LIN {X 0,Y 513.803,Z 636.667,A -85,B 0,C 180,E1 25249.021,E2 25249.021} C_VEL
LIN {X 0,Y 513.812,Z 636.664,A -85,B 0,C 180,E1 25245.53,E2 25245.53} C_VEL
LIN {X 0,Y 513.773,Z 636.668,A -85,B 0,C 180,E1 25244.581,E2 25244.581} C_VEL
LIN {X 0,Y 521.434,Z 663.371,A -85,B 0,C 180,E1 25241.928,E2 25241.928} C_VEL
LIN {X 0,Y 524.036,Z 673.946,A -85,B 0,C 180,E1 25240.926,E2 25240.926} C_VEL
LIN {X 0,Y 522.658,Z 718.938,A -85,B 0,C 180,E1 25237.269,E2 25237.269} C_VEL
LIN {X 0,Y 521.288,Z 761.013,A -85,B 0,C 180,E1 25233.85,E2 25233.85} C_VEL
LIN {X 0,Y 519.996,Z 802.226,A -85,B 0,C 180,E1 25230.503,E2 25230.503} C_VEL
LIN {X 0,Y 519.096,Z 834.822,A -85,B 0,C 180,E1 25227.908,E2 25227.908} C_VEL
LIN {X 0,Y 519.16,Z 847.578,A -85,B 0,C 180,E1 25227.692,E2 25227.692} C_VEL
LIN {X 0,Y 517.25,Z 978.274,A -85,B 0,C 180,E1 25225.563,E2 25225.563} C_VEL
LIN {X 0,Y 517.072,Z 994.179,A -85,B 0,C 180,E1 25225.113,E2 25225.113} C_VEL
LIN {X 0,Y 516.715,Z 1010.152,A -85,B 0,C 180,E1 25224.46,E2 25224.46} C_VEL
LIN {X 0,Y 516.263,Z 1025.12,A -85,B 0,C 180,E1 25223.632,E2 25223.632} C_VEL
LIN {X 0,Y 515.746,Z 1039.216,A -85,B 0,C 180,E1 25222.636,E2 25222.636} C_VEL
LIN {X 0,Y 515.163,Z 1052.41,A -85,B 0,C 180,E1 25221.458,E2 25221.458} C_VEL
LIN {X 0,Y 514.609,Z 1064.521,A -85,B 0,C 180,E1 25220.112,E2 25220.112} C_VEL
LIN {X 0,Y 514.083,Z 1075.294,A -85,B 0,C 180,E1 25218.598,E2 25218.598} C_VEL
LIN {X 0,Y 513.701,Z 1083.812,A -85,B 0,C 180,E1 25217.089,E2 25217.089} C_VEL
LIN {X 0,Y 513.406,Z 1091.297,A -85,B 0,C 180,E1 25215.356,E2 25215.356} C_VEL
LIN {X 0,Y 513.242,Z 1096.383,A -85,B 0,C 180,E1 25213.747,E2 25213.747} C_VEL
LIN {X 0,Y 513.159,Z 1100.181,A -85,B 0,C 180,E1 25211.917,E2 25211.917} C_VEL
LIN {X 0,Y 513.19,Z 1101.973,A -85,B 0,C 180,E1 25210.21,E2 25210.21} C_VEL
LIN {X 0,Y 513.311,Z 1102.014,A -85,B 0,C 180,E1 25208.398,E2 25208.398} C_VEL
LIN {X 0,Y 513.529,Z 1100.384,A -85,B 0,C 180,E1 25206.706,E2 25206.706} C_VEL
LIN {X 0,Y 513.882,Z 1096.719,A -85,B 0,C 180,E1 25204.909,E2 25204.909} C_VEL
LIN {X 0,Y 514.348,Z 1091.471,A -85,B 0,C 180,E1 25203.229,E2 25203.229} C_VEL
LIN {X 0,Y 514.952,Z 1084.154,A -85,B 0,C 180,E1 25201.555,E2 25201.555} C_VEL
LIN {X 0,Y 515.626,Z 1075.956,A -85,B 0,C 180,E1 25200.109,E2 25200.109} C_VEL
LIN {X 0,Y 516.42,Z 1065.525,A -85,B 0,C 180,E1 25198.666,E2 25198.666} C_VEL
LIN {X 0,Y 517.22,Z 1054.065,A -85,B 0,C 180,E1 25197.394,E2 25197.394} C_VEL
LIN {X 0,Y 518.038,Z 1040.208,A -85,B 0,C 180,E1 25196.18,E2 25196.18} C_VEL
LIN {X 0,Y 518.657,Z 1026.603,A -85,B 0,C 180,E1 25195.243,E2 25195.243} C_VEL
LIN {X 0,Y 519.137,Z 1013.166,A -85,B 0,C 180,E1 25194.527,E2 25194.527} C_VEL
LIN {X 0,Y 519.486,Z 999.878,A -85,B 0,C 180,E1 25193.98,E2 25193.98} C_VEL
LIN {X 0,Y 519.702,Z 985.077,A -85,B 0,C 180,E1 25193.528,E2 25193.528} C_VEL
LIN {X 0,Y 520.188,Z 943.34,A -85,B 0,C 180,E1 25192.784,E2 25192.784} C_VEL
LIN {X 0,Y 522.879,Z 843.141,A -85,B 0,C 180,E1 25191.004,E2 25191.004} C_VEL
LIN {X 0,Y 523.363,Z 837.807,A -85,B 0,C 180,E1 25190.596,E2 25190.596} C_VEL
LIN {X 0,Y 524.872,Z 795.815,A -85,B 0,C 180,E1 25187.231,E2 25187.231} C_VEL
LIN {X 0,Y 526.347,Z 751.412,A -85,B 0,C 180,E1 25183.726,E2 25183.726} C_VEL
LIN {X 0,Y 527.629,Z 711.745,A -85,B 0,C 180,E1 25180.63,E2 25180.63} C_VEL
LIN {X 0,Y 528.648,Z 676.247,A -85,B 0,C 180,E1 25177.888,E2 25177.888} C_VEL
LIN {X 0,Y 524.106,Z 661.406,A -85,B 0,C 180,E1 25176.306,E2 25176.306} C_VEL
LIN {X 0,Y 518.577,Z 647.638,A -85,B 0,C 180,E1 25174.654,E2 25174.654} C_VEL
LIN {X 0,Y 515.244,Z 640.334,A -85,B 0,C 180,E1 25173.705,E2 25173.705} C_VEL
LIN {X 0,Y 513.838,Z 636.878,A -85,B 0,C 180,E1 25173.27,E2 25173.27} C_VEL
LIN {X 0,Y 513.821,Z 636.667,A -85,B 0,C 180,E1 25169.732,E2 25169.732} C_VEL
LIN {X 0,Y 513.795,Z 636.668,A -85,B 0,C 180,E1 25166.178,E2 25166.178} C_VEL
LIN {X 0,Y 513.774,Z 636.672,A -85,B 0,C 180,E1 25162.744,E2 25162.744} C_VEL
LIN {X 0,Y 513.814,Z 636.668,A -85,B 0,C 180,E1 25159.312,E2 25159.312} C_VEL
LIN {X 0,Y 513.792,Z 636.669,A -85,B 0,C 180,E1 25155.835,E2 25155.835} C_VEL
LIN {X 0,Y 513.811,Z 636.697,A -85,B 0,C 180,E1 25153.08,E2 25153.08} C_VEL
LIN {X 0,Y 521.914,Z 661.069,A -85,B 0,C 180,E1 25149.638,E2 25149.638} C_VEL
LIN {X 0,Y 527.08,Z 677.245,A -85,B 0,C 180,E1 25147.513,E2 25147.513} C_VEL
LIN {X 0,Y 536.092,Z 695.93,A -85,B 0,C 180,E1 25146.509,E2 25146.509} C_VEL
LIN {X 0,Y 541.946,Z 727.791,A -85,B 0,C 180,E1 25145.51,E2 25145.51} C_VEL
LIN {X 0,Y 534.149,Z 956.257,A -85,B 0,C 180,E1 25141.827,E2 25141.827} C_VEL
LIN {X 0,Y 532.929,Z 987.725,A -85,B 0,C 180,E1 25141.267,E2 25141.267} C_VEL
LIN {X 0,Y 531.526,Z 1010.263,A -85,B 0,C 180,E1 25140.678,E2 25140.678} C_VEL
LIN {X 0,Y 529.841,Z 1032.153,A -85,B 0,C 180,E1 25139.91,E2 25139.91} C_VEL
LIN {X 0,Y 527.905,Z 1053.634,A -85,B 0,C 180,E1 25138.945,E2 25138.945} C_VEL
LIN {X 0,Y 525.899,Z 1073.923,A -85,B 0,C 180,E1 25137.829,E2 25137.829} C_VEL
LIN {X 0,Y 523.792,Z 1093.66,A -85,B 0,C 180,E1 25136.53,E2 25136.53} C_VEL
LIN {X 0,Y 521.699,Z 1112.467,A -85,B 0,C 180,E1 25135.058,E2 25135.058} C_VEL
LIN {X 0,Y 519.71,Z 1129.674,A -85,B 0,C 180,E1 25133.467,E2 25133.467} C_VEL
LIN {X 0,Y 517.788,Z 1146.563,A -85,B 0,C 180,E1 25131.642,E2 25131.642} C_VEL
LIN {X 0,Y 516.219,Z 1161.109,A -85,B 0,C 180,E1 25129.812,E2 25129.812} C_VEL
LIN {X 0,Y 514.799,Z 1174.994,A -85,B 0,C 180,E1 25127.753,E2 25127.753} C_VEL
LIN {X 0,Y 513.736,Z 1186.732,A -85,B 0,C 180,E1 25125.694,E2 25125.694} C_VEL
LIN {X 0,Y 512.948,Z 1197.192,A -85,B 0,C 180,E1 25123.526,E2 25123.526} C_VEL
LIN {X 0,Y 512.434,Z 1205.782,A -85,B 0,C 180,E1 25121.364,E2 25121.364} C_VEL
LIN {X 0,Y 512.144,Z 1212.979,A -85,B 0,C 180,E1 25119.097,E2 25119.097} C_VEL
LIN {X 0,Y 512.011,Z 1218.543,A -85,B 0,C 180,E1 25116.84,E2 25116.84} C_VEL
LIN {X 0,Y 511.993,Z 1222.401,A -85,B 0,C 180,E1 25114.591,E2 25114.591} C_VEL
LIN {X 0,Y 512.019,Z 1224.805,A -85,B 0,C 180,E1 25112.237,E2 25112.237} C_VEL
LIN {X 0,Y 512.036,Z 1225.575,A -85,B 0,C 180,E1 25109.998,E2 25109.998} C_VEL
LIN {X 0,Y 512.022,Z 1224.636,A -85,B 0,C 180,E1 25107.648,E2 25107.648} C_VEL
LIN {X 0,Y 511.996,Z 1222.078,A -85,B 0,C 180,E1 25105.294,E2 25105.294} C_VEL
LIN {X 0,Y 512.023,Z 1218.018,A -85,B 0,C 180,E1 25103.044,E2 25103.044} C_VEL
LIN {X 0,Y 512.153,Z 1212.299,A -85,B 0,C 180,E1 25100.786,E2 25100.786} C_VEL
LIN {X 0,Y 512.446,Z 1204.906,A -85,B 0,C 180,E1 25098.519,E2 25098.519} C_VEL
LIN {X 0,Y 512.962,Z 1196.072,A -85,B 0,C 180,E1 25096.356,E2 25096.356} C_VEL
LIN {X 0,Y 513.803,Z 1184.785,A -85,B 0,C 180,E1 25094.073,E2 25094.073} C_VEL
LIN {X 0,Y 514.88,Z 1172.684,A -85,B 0,C 180,E1 25092.013,E2 25092.013} C_VEL
LIN {X 0,Y 516.229,Z 1159.214,A -85,B 0,C 180,E1 25090.067,E2 25090.067} C_VEL
LIN {X 0,Y 517.86,Z 1143.949,A -85,B 0,C 180,E1 25088.179,E2 25088.179} C_VEL
LIN {X 0,Y 519.798,Z 1126.723,A -85,B 0,C 180,E1 25086.354,E2 25086.354} C_VEL
LIN {X 0,Y 521.898,Z 1108.529,A -85,B 0,C 180,E1 25084.706,E2 25084.706} C_VEL
LIN {X 0,Y 524.159,Z 1088.605,A -85,B 0,C 180,E1 25083.181,E2 25083.181} C_VEL
LIN {X 0,Y 526.34,Z 1068.631,A -85,B 0,C 180,E1 25081.891,E2 25081.891} C_VEL
LIN {X 0,Y 528.717,Z 1045.94,A -85,B 0,C 180,E1 25080.671,E2 25080.671} C_VEL
LIN {X 0,Y 530.982,Z 1022.681,A -85,B 0,C 180,E1 25079.658,E2 25079.658} C_VEL
LIN {X 0,Y 533.053,Z 999.229,A -85,B 0,C 180,E1 25078.855,E2 25078.855} C_VEL
LIN {X 0,Y 534.916,Z 974.798,A -85,B 0,C 180,E1 25078.231,E2 25078.231} C_VEL
LIN {X 0,Y 540.351,Z 876.827,A -85,B 0,C 180,E1 25076.311,E2 25076.311} C_VEL
LIN {X 0,Y 546.67,Z 793.592,A -85,B 0,C 180,E1 25074.546,E2 25074.546} C_VEL
LIN {X 0,Y 552.856,Z 728.302,A -85,B 0,C 180,E1 25073.075,E2 25073.075} C_VEL
LIN {X 0,Y 551.722,Z 708.154,A -85,B 0,C 180,E1 25072.093,E2 25072.093} C_VEL
LIN {X 0,Y 551.305,Z 705.302,A -85,B 0,C 180,E1 25071.9,E2 25071.9} C_VEL
LIN {X 0,Y 548.013,Z 696.634,A -85,B 0,C 180,E1 25070.889,E2 25070.889} C_VEL
LIN {X 0,Y 544.817,Z 689.432,A -85,B 0,C 180,E1 25069.774,E2 25069.774} C_VEL
LIN {X 0,Y 541.478,Z 682.343,A -85,B 0,C 180,E1 25068.301,E2 25068.301} C_VEL
LIN {X 0,Y 539.164,Z 677.441,A -85,B 0,C 180,E1 25066.712,E2 25066.712} C_VEL
LIN {X 0,Y 538.11,Z 674.401,A -85,B 0,C 180,E1 25064.92,E2 25064.92} C_VEL
LIN {X 0,Y 538.584,Z 674.12,A -85,B 0,C 180,E1 25063.388,E2 25063.388} C_VEL
LIN {X 0,Y 539.903,Z 674.802,A -85,B 0,C 180,E1 25062.2,E2 25062.2} C_VEL
LIN {X 0,Y 542.161,Z 677.465,A -85,B 0,C 180,E1 25060.873,E2 25060.873} C_VEL
LIN {X 0,Y 545.573,Z 681.913,A -85,B 0,C 180,E1 25059.493,E2 25059.493} C_VEL
LIN {X 0,Y 548.979,Z 687.07,A -85,B 0,C 180,E1 25058.408,E2 25058.408} C_VEL
LIN {X 0,Y 553.667,Z 694.94,A -85,B 0,C 180,E1 25057.167,E2 25057.167} C_VEL
LIN {X 0,Y 555.184,Z 698.399,A -85,B 0,C 180,E1 25056.777,E2 25056.777} C_VEL
LIN {X 0,Y 546.82,Z 780.12,A -85,B 0,C 180,E1 25054.935,E2 25054.935} C_VEL
LIN {X 0,Y 540.554,Z 860.314,A -85,B 0,C 180,E1 25053.231,E2 25053.231} C_VEL
LIN {X 0,Y 535.689,Z 943.992,A -85,B 0,C 180,E1 25051.546,E2 25051.546} C_VEL
LIN {X 0,Y 534.196,Z 966.908,A -85,B 0,C 180,E1 25050.888,E2 25050.888} C_VEL
LIN {X 0,Y 532.354,Z 989.55,A -85,B 0,C 180,E1 25050.032,E2 25050.032} C_VEL
LIN {X 0,Y 530.289,Z 1011.418,A -85,B 0,C 180,E1 25048.987,E2 25048.987} C_VEL
LIN {X 0,Y 528.165,Z 1031.475,A -85,B 0,C 180,E1 25047.82,E2 25047.82} C_VEL
LIN {X 0,Y 525.838,Z 1051.668,A -85,B 0,C 180,E1 25046.411,E2 25046.411} C_VEL
LIN {X 0,Y 523.606,Z 1069.983,A -85,B 0,C 180,E1 25044.895,E2 25044.895} C_VEL
LIN {X 0,Y 521.408,Z 1087.263,A -85,B 0,C 180,E1 25043.211,E2 25043.211} C_VEL
LIN {X 0,Y 519.411,Z 1102.479,A -85,B 0,C 180,E1 25041.456,E2 25041.456} C_VEL
LIN {X 0,Y 517.567,Z 1116.812,A -85,B 0,C 180,E1 25039.527,E2 25039.527} C_VEL
LIN {X 0,Y 516.045,Z 1129.207,A -85,B 0,C 180,E1 25037.577,E2 25037.577} C_VEL
LIN {X 0,Y 514.714,Z 1140.622,A -85,B 0,C 180,E1 25035.437,E2 25035.437} C_VEL
LIN {X 0,Y 513.724,Z 1150.177,A -85,B 0,C 180,E1 25033.28,E2 25033.28} C_VEL
LIN {X 0,Y 512.988,Z 1158.434,A -85,B 0,C 180,E1 25031.014,E2 25031.014} C_VEL
LIN {X 0,Y 512.518,Z 1164.925,A -85,B 0,C 180,E1 25028.755,E2 25028.755} C_VEL
LIN {X 0,Y 512.245,Z 1169.75,A -85,B 0,C 180,E1 25026.503,E2 25026.503} C_VEL
LIN {X 0,Y 512.098,Z 1173.26,A -85,B 0,C 180,E1 25024.145,E2 25024.145} C_VEL
LIN {X 0,Y 512.043,Z 1175.029,A -85,B 0,C 180,E1 25021.905,E2 25021.905} C_VEL
LIN {X 0,Y 512.033,Z 1175.327,A -85,B 0,C 180,E1 25019.443,E2 25019.443} C_VEL
LIN {X 0,Y 512.047,Z 1174.044,A -85,B 0,C 180,E1 25017.092,E2 25017.092} C_VEL
LIN {X 0,Y 512.106,Z 1171.071,A -85,B 0,C 180,E1 25014.737,E2 25014.737} C_VEL
LIN {X 0,Y 512.267,Z 1166.46,A -85,B 0,C 180,E1 25012.375,E2 25012.375} C_VEL
LIN {X 0,Y 512.584,Z 1160.455,A -85,B 0,C 180,E1 25010.099,E2 25010.099} C_VEL
LIN {X 0,Y 513.095,Z 1152.768,A -85,B 0,C 180,E1 25007.853,E2 25007.853} C_VEL
LIN {X 0,Y 513.884,Z 1143.176,A -85,B 0,C 180,E1 25005.581,E2 25005.581} C_VEL
LIN {X 0,Y 514.955,Z 1132.184,A -85,B 0,C 180,E1 25003.418,E2 25003.418} C_VEL
LIN {X 0,Y 516.293,Z 1119.773,A -85,B 0,C 180,E1 25001.367,E2 25001.367} C_VEL
LIN {X 0,Y 517.862,Z 1105.912,A -85,B 0,C 180,E1 24999.43,E2 24999.43} C_VEL
LIN {X 0,Y 519.775,Z 1089.684,A -85,B 0,C 180,E1 24997.495,E2 24997.495} C_VEL
LIN {X 0,Y 521.714,Z 1073.28,A -85,B 0,C 180,E1 24995.823,E2 24995.823} C_VEL
LIN {X 0,Y 523.789,Z 1055.294,A -85,B 0,C 180,E1 24994.269,E2 24994.269} C_VEL
LIN {X 0,Y 525.791,Z 1036.692,A -85,B 0,C 180,E1 24992.909,E2 24992.909} C_VEL
LIN {X 0,Y 527.907,Z 1015.639,A -85,B 0,C 180,E1 24991.617,E2 24991.617} C_VEL
LIN {X 0,Y 529.772,Z 994.948,A -85,B 0,C 180,E1 24990.571,E2 24990.571} C_VEL
LIN {X 0,Y 531.447,Z 973.249,A -85,B 0,C 180,E1 24989.692,E2 24989.692} C_VEL
LIN {X 0,Y 532.803,Z 951.506,A -85,B 0,C 180,E1 24989.016,E2 24989.016} C_VEL
LIN {X 0,Y 533.895,Z 928.174,A -85,B 0,C 180,E1 24988.49,E2 24988.49} C_VEL
LIN {X 0,Y 541.791,Z 696.963,A -85,B 0,C 180,E1 24984.767,E2 24984.767} C_VEL
LIN {X 0,Y 541.921,Z 688.048,A -85,B 0,C 180,E1 24984.609,E2 24984.609} C_VEL
LIN {X 0,Y 531.027,Z 667.774,A -85,B 0,C 180,E1 24983.471,E2 24983.471} C_VEL
LIN {X 0,Y 515.293,Z 640.454,A -85,B 0,C 180,E1 24981.78,E2 24981.78} C_VEL
LIN {X 0,Y 513.852,Z 637.155,A -85,B 0,C 180,E1 24981.602,E2 24981.602} C_VEL
LIN {X 0,Y 513.777,Z 636.668,A -85,B 0,C 180,E1 24981.567,E2 24981.567} C_VEL
LIN {X 0,Y 513.801,Z 636.662,A -85,B 0,C 180,E1 24978.023,E2 24978.023} C_VEL
LIN {X 0,Y 513.783,Z 636.666,A -85,B 0,C 180,E1 24974.584,E2 24974.584} C_VEL
LIN {X 0,Y 513.74,Z 636.674,A -85,B 0,C 180,E1 24971.135,E2 24971.135} C_VEL
LIN {X 0,Y 513.761,Z 636.669,A -85,B 0,C 180,E1 24967.671,E2 24967.671} C_VEL
LIN {X 0,Y 513.807,Z 636.667,A -85,B 0,C 180,E1 24964.358,E2 24964.358} C_VEL
LIN {X 0,Y 513.811,Z 636.67,A -85,B 0,C 180,E1 24960.785,E2 24960.785} C_VEL
LIN {X 0,Y 513.813,Z 636.67,A -85,B 0,C 180,E1 24957.341,E2 24957.341} C_VEL
LIN {X 0,Y 513.78,Z 636.672,A -85,B 0,C 180,E1 24953.88,E2 24953.88} C_VEL
LIN {X 0,Y 513.757,Z 636.674,A -85,B 0,C 180,E1 24951.238,E2 24951.238} C_VEL
LIN {X 0,Y 512.74,Z 636.805,A -85,B 0,C 180,E1 24950.38,E2 24950.38} C_VEL
LIN {X 0,Y 506.308,Z 637.601,A -85,B 0,C 180,E1 24947.902,E2 24947.902} C_VEL
LIN {X 0,Y 505.852,Z 637.654,A -85,B 0,C 180,E1 24947.336,E2 24947.336} C_VEL
LIN {X 0,Y 505.87,Z 637.646,A -85,B 0,C 180,E1 24943.955,E2 24943.955} C_VEL
LIN {X 0,Y 505.857,Z 637.656,A -85,B 0,C 180,E1 24940.364,E2 24940.364} C_VEL
LIN {X 0,Y 505.872,Z 637.651,A -85,B 0,C 180,E1 24936.926,E2 24936.926} C_VEL
LIN {X 0,Y 505.819,Z 637.655,A -85,B 0,C 180,E1 24933.401,E2 24933.401} C_VEL
LIN {X 0,Y 505.815,Z 637.659,A -85,B 0,C 180,E1 24930.002,E2 24930.002} C_VEL
LIN {X 0,Y 505.849,Z 637.643,A -85,B 0,C 180,E1 24926.489,E2 24926.489} C_VEL
LIN {X 0,Y 505.864,Z 637.652,A -85,B 0,C 180,E1 24922.962,E2 24922.962} C_VEL
LIN {X 0,Y 505.821,Z 637.644,A -85,B 0,C 180,E1 24919.524,E2 24919.524} C_VEL
LIN {X 0,Y 505.805,Z 637.661,A -85,B 0,C 180,E1 24916.046,E2 24916.046} C_VEL
LIN {X 0,Y 505.863,Z 637.655,A -85,B 0,C 180,E1 24912.636,E2 24912.636} C_VEL
LIN {X 0,Y 505.863,Z 637.656,A -85,B 0,C 180,E1 24909.16,E2 24909.16} C_VEL
LIN {X 0,Y 505.865,Z 637.656,A -85,B 0,C 180,E1 24905.602,E2 24905.602} C_VEL
LIN {X 0,Y 505.878,Z 637.654,A -85,B 0,C 180,E1 24902.062,E2 24902.062} C_VEL
LIN {X 0,Y 505.801,Z 637.662,A -85,B 0,C 180,E1 24898.809,E2 24898.809} C_VEL
LIN {X 0,Y 505.806,Z 637.661,A -85,B 0,C 180,E1 24895.299,E2 24895.299} C_VEL
LIN {X 0,Y 505.863,Z 637.654,A -85,B 0,C 180,E1 24891.871,E2 24891.871} C_VEL
LIN {X 0,Y 505.862,Z 637.655,A -85,B 0,C 180,E1 24888.387,E2 24888.387} C_VEL
LIN {X 0,Y 505.864,Z 637.769,A -85,B 0,C 180,E1 24884.911,E2 24884.911} C_VEL
LIN {X 0,Y 513.499,Z 664.113,A -85,B 0,C 180,E1 24882.277,E2 24882.277} C_VEL
LIN {X 0,Y 516.484,Z 675.76,A -85,B 0,C 180,E1 24881.145,E2 24881.145} C_VEL
LIN {X 0,Y 515.073,Z 719.612,A -85,B 0,C 180,E1 24877.553,E2 24877.553} C_VEL
LIN {X 0,Y 513.653,Z 761.956,A -85,B 0,C 180,E1 24874.095,E2 24874.095} C_VEL
LIN {X 0,Y 512.326,Z 802.972,A -85,B 0,C 180,E1 24870.749,E2 24870.749} C_VEL
LIN {X 0,Y 511.378,Z 835.651,A -85,B 0,C 180,E1 24868.126,E2 24868.126} C_VEL
LIN {X 0,Y 511.291,Z 854.106,A -85,B 0,C 180,E1 24867.808,E2 24867.808} C_VEL
LIN {X 0,Y 509.418,Z 979.153,A -85,B 0,C 180,E1 24865.732,E2 24865.732} C_VEL
LIN {X 0,Y 509.236,Z 994.955,A -85,B 0,C 180,E1 24865.278,E2 24865.278} C_VEL
LIN {X 0,Y 508.867,Z 1010.953,A -85,B 0,C 180,E1 24864.615,E2 24864.615} C_VEL
LIN {X 0,Y 508.402,Z 1025.957,A -85,B 0,C 180,E1 24863.774,E2 24863.774} C_VEL
LIN {X 0,Y 507.875,Z 1039.878,A -85,B 0,C 180,E1 24862.778,E2 24862.778} C_VEL
LIN {X 0,Y 507.294,Z 1052.71,A -85,B 0,C 180,E1 24861.625,E2 24861.625} C_VEL
LIN {X 0,Y 506.717,Z 1064.951,A -85,B 0,C 180,E1 24860.259,E2 24860.259} C_VEL
LIN {X 0,Y 506.188,Z 1075.466,A -85,B 0,C 180,E1 24858.78,E2 24858.78} C_VEL
LIN {X 0,Y 505.787,Z 1084.177,A -85,B 0,C 180,E1 24857.247,E2 24857.247} C_VEL
LIN {X 0,Y 505.479,Z 1091.481,A -85,B 0,C 180,E1 24855.572,E2 24855.572} C_VEL
LIN {X 0,Y 505.299,Z 1097.053,A -85,B 0,C 180,E1 24853.85,E2 24853.85} C_VEL
LIN {X 0,Y 505.208,Z 1101.155,A -85,B 0,C 180,E1 24851.875,E2 24851.875} C_VEL
LIN {X 0,Y 505.249,Z 1102.957,A -85,B 0,C 180,E1 24850.142,E2 24850.142} C_VEL
LIN {X 0,Y 505.386,Z 1103.004,A -85,B 0,C 180,E1 24848.301,E2 24848.301} C_VEL
LIN {X 0,Y 505.628,Z 1101.365,A -85,B 0,C 180,E1 24846.583,E2 24846.583} C_VEL
LIN {X 0,Y 506.014,Z 1097.685,A -85,B 0,C 180,E1 24844.758,E2 24844.758} C_VEL
LIN {X 0,Y 506.516,Z 1092.403,A -85,B 0,C 180,E1 24843.053,E2 24843.053} C_VEL
LIN {X 0,Y 507.17,Z 1085.067,A -85,B 0,C 180,E1 24841.353,E2 24841.353} C_VEL
LIN {X 0,Y 507.924,Z 1076.532,A -85,B 0,C 180,E1 24839.835,E2 24839.835} C_VEL
LIN {X 0,Y 508.825,Z 1065.529,A -85,B 0,C 180,E1 24838.308,E2 24838.308} C_VEL
LIN {X 0,Y 509.676,Z 1053.728,A -85,B 0,C 180,E1 24837.018,E2 24837.018} C_VEL
LIN {X 0,Y 510.505,Z 1040.242,A -85,B 0,C 180,E1 24835.842,E2 24835.842} C_VEL
LIN {X 0,Y 511.202,Z 1025.357,A -85,B 0,C 180,E1 24834.836,E2 24834.836} C_VEL
LIN {X 0,Y 511.664,Z 1012.389,A -85,B 0,C 180,E1 24834.165,E2 24834.165} C_VEL
LIN {X 0,Y 512.003,Z 1000.141,A -85,B 0,C 180,E1 24833.663,E2 24833.663} C_VEL
LIN {X 0,Y 512.227,Z 985.675,A -85,B 0,C 180,E1 24833.219,E2 24833.219} C_VEL
LIN {X 0,Y 512.765,Z 944.371,A -85,B 0,C 180,E1 24832.462,E2 24832.462} C_VEL
LIN {X 0,Y 515.597,Z 844.473,A -85,B 0,C 180,E1 24830.651,E2 24830.651} C_VEL
LIN {X 0,Y 516.081,Z 840.687,A -85,B 0,C 180,E1 24830.365,E2 24830.365} C_VEL
LIN {X 0,Y 517.535,Z 801.653,A -85,B 0,C 180,E1 24827.217,E2 24827.217} C_VEL
LIN {X 0,Y 519.119,Z 760.021,A -85,B 0,C 180,E1 24823.895,E2 24823.895} C_VEL
LIN {X 0,Y 520.544,Z 719.711,A -85,B 0,C 180,E1 24820.706,E2 24820.706} C_VEL
LIN {X 0,Y 521.881,Z 679.231,A -85,B 0,C 180,E1 24817.526,E2 24817.526} C_VEL
LIN {X 0,Y 517.477,Z 664.782,A -85,B 0,C 180,E1 24815.937,E2 24815.937} C_VEL
LIN {X 0,Y 511.422,Z 649.701,A -85,B 0,C 180,E1 24814.068,E2 24814.068} C_VEL
LIN {X 0,Y 507.417,Z 641.49,A -85,B 0,C 180,E1 24812.92,E2 24812.92} C_VEL
LIN {X 0,Y 505.913,Z 638.115,A -85,B 0,C 180,E1 24812.451,E2 24812.451} C_VEL
LIN {X 0,Y 505.842,Z 637.662,A -85,B 0,C 180,E1 24812.383,E2 24812.383} C_VEL
LIN {X 0,Y 505.867,Z 637.657,A -85,B 0,C 180,E1 24808.809,E2 24808.809} C_VEL
LIN {X 0,Y 505.869,Z 637.654,A -85,B 0,C 180,E1 24805.109,E2 24805.109} C_VEL
LIN {X 0,Y 505.879,Z 637.655,A -85,B 0,C 180,E1 24801.491,E2 24801.491} C_VEL
LIN {X 0,Y 505.855,Z 637.659,A -85,B 0,C 180,E1 24797.925,E2 24797.925} C_VEL
LIN {X 0,Y 505.836,Z 637.653,A -85,B 0,C 180,E1 24794.47,E2 24794.47} C_VEL
LIN {X 0,Y 505.878,Z 637.765,A -85,B 0,C 180,E1 24793.612,E2 24793.612} C_VEL
LIN {X 0,Y 513.797,Z 661.454,A -85,B 0,C 180,E1 24790.194,E2 24790.194} C_VEL
LIN {X 0,Y 518.836,Z 677.056,A -85,B 0,C 180,E1 24788.113,E2 24788.113} C_VEL
LIN {X 0,Y 529.687,Z 699.314,A -85,B 0,C 180,E1 24786.89,E2 24786.89} C_VEL
LIN {X 0,Y 535.088,Z 729.102,A -85,B 0,C 180,E1 24785.938,E2 24785.938} C_VEL
LIN {X 0,Y 526.816,Z 960.456,A -85,B 0,C 180,E1 24782.137,E2 24782.137} C_VEL
LIN {X 0,Y 525.646,Z 988.208,A -85,B 0,C 180,E1 24781.623,E2 24781.623} C_VEL
LIN {X 0,Y 524.16,Z 1010.945,A -85,B 0,C 180,E1 24781.011,E2 24781.011} C_VEL
LIN {X 0,Y 522.404,Z 1032.934,A -85,B 0,C 180,E1 24780.222,E2 24780.222} C_VEL
LIN {X 0,Y 520.348,Z 1054.824,A -85,B 0,C 180,E1 24779.212,E2 24779.212} C_VEL
LIN {X 0,Y 518.277,Z 1074.826,A -85,B 0,C 180,E1 24778.08,E2 24778.08} C_VEL
LIN {X 0,Y 516.028,Z 1095.036,A -85,B 0,C 180,E1 24776.711,E2 24776.711} C_VEL
LIN {X 0,Y 513.883,Z 1113.63,A -85,B 0,C 180,E1 24775.219,E2 24775.219} C_VEL
LIN {X 0,Y 511.784,Z 1131.234,A -85,B 0,C 180,E1 24773.547,E2 24773.547} C_VEL
LIN {X 0,Y 509.877,Z 1147.363,A -85,B 0,C 180,E1 24771.753,E2 24771.753} C_VEL
LIN {X 0,Y 508.178,Z 1162.559,A -85,B 0,C 180,E1 24769.779,E2 24769.779} C_VEL
LIN {X 0,Y 506.824,Z 1175.574,A -85,B 0,C 180,E1 24767.804,E2 24767.804} C_VEL
LIN {X 0,Y 505.713,Z 1187.47,A -85,B 0,C 180,E1 24765.653,E2 24765.653} C_VEL
LIN {X 0,Y 504.907,Z 1197.952,A -85,B 0,C 180,E1 24763.395,E2 24763.395} C_VEL
LIN {X 0,Y 504.393,Z 1206.729,A -85,B 0,C 180,E1 24761.101,E2 24761.101} C_VEL
LIN {X 0,Y 504.123,Z 1213.695,A -85,B 0,C 180,E1 24758.783,E2 24758.783} C_VEL
LIN {X 0,Y 504.016,Z 1219.129,A -85,B 0,C 180,E1 24756.377,E2 24756.377} C_VEL
LIN {X 0,Y 504.01,Z 1222.726,A -85,B 0,C 180,E1 24754.094,E2 24754.094} C_VEL
LIN {X 0,Y 504.03,Z 1224.648,A -85,B 0,C 180,E1 24751.817,E2 24751.817} C_VEL
LIN {X 0,Y 504.031,Z 1225.075,A -85,B 0,C 180,E1 24749.43,E2 24749.43} C_VEL
LIN {X 0,Y 504.019,Z 1223.996,A -85,B 0,C 180,E1 24747.269,E2 24747.269} C_VEL
LIN {X 0,Y 504,Z 1221.154,A -85,B 0,C 180,E1 24744.877,E2 24744.877} C_VEL
LIN {X 0,Y 504.045,Z 1216.907,A -85,B 0,C 180,E1 24742.59,E2 24742.59} C_VEL
LIN {X 0,Y 504.198,Z 1210.846,A -85,B 0,C 180,E1 24740.277,E2 24740.277} C_VEL
LIN {X 0,Y 504.58,Z 1202.727,A -85,B 0,C 180,E1 24737.873,E2 24737.873} C_VEL
LIN {X 0,Y 505.184,Z 1193.605,A -85,B 0,C 180,E1 24735.675,E2 24735.675} C_VEL
LIN {X 0,Y 506.105,Z 1182.472,A -85,B 0,C 180,E1 24733.47,E2 24733.47} C_VEL
LIN {X 0,Y 507.303,Z 1169.962,A -85,B 0,C 180,E1 24731.378,E2 24731.378} C_VEL
LIN {X 0,Y 508.796,Z 1156.181,A -85,B 0,C 180,E1 24729.403,E2 24729.403} C_VEL
LIN {X 0,Y 510.6,Z 1140.498,A -85,B 0,C 180,E1 24727.489,E2 24727.489} C_VEL
LIN {X 0,Y 512.594,Z 1123.851,A -85,B 0,C 180,E1 24725.749,E2 24725.749} C_VEL
LIN {X 0,Y 514.903,Z 1104.786,A -85,B 0,C 180,E1 24724.043,E2 24724.043} C_VEL
LIN {X 0,Y 517.263,Z 1085.318,A -85,B 0,C 180,E1 24722.562,E2 24722.562} C_VEL
LIN {X 0,Y 519.647,Z 1064.758,A -85,B 0,C 180,E1 24721.245,E2 24721.245} C_VEL
LIN {X 0,Y 521.968,Z 1043.776,A -85,B 0,C 180,E1 24720.127,E2 24720.127} C_VEL
LIN {X 0,Y 524.373,Z 1020.303,A -85,B 0,C 180,E1 24719.103,E2 24719.103} C_VEL
LIN {X 0,Y 526.686,Z 995.904,A -85,B 0,C 180,E1 24718.276,E2 24718.276} C_VEL
LIN {X 0,Y 528.605,Z 971.57,A -85,B 0,C 180,E1 24717.658,E2 24717.658} C_VEL
LIN {X 0,Y 534.336,Z 878.241,A -85,B 0,C 180,E1 24715.762,E2 24715.762} C_VEL
LIN {X 0,Y 540.95,Z 798.481,A -85,B 0,C 180,E1 24714.015,E2 24714.015} C_VEL
LIN {X 0,Y 548.015,Z 730.026,A -85,B 0,C 180,E1 24712.427,E2 24712.427} C_VEL
LIN {X 0,Y 547.276,Z 710.873,A -85,B 0,C 180,E1 24711.454,E2 24711.454} C_VEL
LIN {X 0,Y 544.725,Z 703.308,A -85,B 0,C 180,E1 24710.571,E2 24710.571} C_VEL
LIN {X 0,Y 541.798,Z 696.206,A -85,B 0,C 180,E1 24709.456,E2 24709.456} C_VEL
LIN {X 0,Y 538.924,Z 689.492,A -85,B 0,C 180,E1 24708.031,E2 24708.031} C_VEL
LIN {X 0,Y 536.856,Z 684.774,A -85,B 0,C 180,E1 24706.43,E2 24706.43} C_VEL
LIN {X 0,Y 536.161,Z 681.932,A -85,B 0,C 180,E1 24704.676,E2 24704.676} C_VEL
LIN {X 0,Y 536.855,Z 681.962,A -85,B 0,C 180,E1 24703.104,E2 24703.104} C_VEL
LIN {X 0,Y 538.101,Z 682.802,A -85,B 0,C 180,E1 24702.067,E2 24702.067} C_VEL
LIN {X 0,Y 540.539,Z 686.021,A -85,B 0,C 180,E1 24700.674,E2 24700.674} C_VEL
LIN {X 0,Y 542.92,Z 689.22,A -85,B 0,C 180,E1 24699.706,E2 24699.706} C_VEL
LIN {X 0,Y 546.324,Z 694.618,A -85,B 0,C 180,E1 24698.559,E2 24698.559} C_VEL
LIN {X 0,Y 550.346,Z 701.957,A -85,B 0,C 180,E1 24697.421,E2 24697.421} C_VEL
LIN {X 0,Y 542.22,Z 774.734,A -85,B 0,C 180,E1 24695.709,E2 24695.709} C_VEL
LIN {X 0,Y 535.355,Z 852.177,A -85,B 0,C 180,E1 24693.994,E2 24693.994} C_VEL
LIN {X 0,Y 529.235,Z 945.487,A -85,B 0,C 180,E1 24692.036,E2 24692.036} C_VEL
LIN {X 0,Y 527.587,Z 968.465,A -85,B 0,C 180,E1 24691.35,E2 24691.35} C_VEL
LIN {X 0,Y 525.596,Z 991.208,A -85,B 0,C 180,E1 24690.465,E2 24690.465} C_VEL
LIN {X 0,Y 523.305,Z 1013.867,A -85,B 0,C 180,E1 24689.349,E2 24689.349} C_VEL
LIN {X 0,Y 520.969,Z 1034.335,A -85,B 0,C 180,E1 24688.113,E2 24688.113} C_VEL
LIN {X 0,Y 518.549,Z 1053.908,A -85,B 0,C 180,E1 24686.7,E2 24686.7} C_VEL
LIN {X 0,Y 516.118,Z 1072.51,A -85,B 0,C 180,E1 24685.107,E2 24685.107} C_VEL
LIN {X 0,Y 513.818,Z 1089.523,A -85,B 0,C 180,E1 24683.392,E2 24683.392} C_VEL
LIN {X 0,Y 511.663,Z 1105.195,A -85,B 0,C 180,E1 24681.533,E2 24681.533} C_VEL
LIN {X 0,Y 509.673,Z 1119.759,A -85,B 0,C 180,E1 24679.484,E2 24679.484} C_VEL
LIN {X 0,Y 508.032,Z 1132.241,A -85,B 0,C 180,E1 24677.409,E2 24677.409} C_VEL
LIN {X 0,Y 506.751,Z 1142.842,A -85,B 0,C 180,E1 24675.334,E2 24675.334} C_VEL
LIN {X 0,Y 505.743,Z 1152.098,A -85,B 0,C 180,E1 24673.144,E2 24673.144} C_VEL
LIN {X 0,Y 504.999,Z 1160.011,A -85,B 0,C 180,E1 24670.844,E2 24670.844} C_VEL
LIN {X 0,Y 504.526,Z 1166.326,A -85,B 0,C 180,E1 24668.526,E2 24668.526} C_VEL
LIN {X 0,Y 504.241,Z 1171.046,A -85,B 0,C 180,E1 24666.149,E2 24666.149} C_VEL
LIN {X 0,Y 504.104,Z 1174.151,A -85,B 0,C 180,E1 24663.755,E2 24663.755} C_VEL
LIN {X 0,Y 504.058,Z 1175.709,A -85,B 0,C 180,E1 24661.366,E2 24661.366} C_VEL
LIN {X 0,Y 504.044,Z 1175.632,A -85,B 0,C 180,E1 24659.093,E2 24659.093} C_VEL
LIN {X 0,Y 504.061,Z 1173.903,A -85,B 0,C 180,E1 24656.591,E2 24656.591} C_VEL
LIN {X 0,Y 504.141,Z 1170.647,A -85,B 0,C 180,E1 24654.197,E2 24654.197} C_VEL
LIN {X 0,Y 504.324,Z 1165.903,A -85,B 0,C 180,E1 24651.91,E2 24651.91} C_VEL
LIN {X 0,Y 504.71,Z 1159.214,A -85,B 0,C 180,E1 24649.501,E2 24649.501} C_VEL
LIN {X 0,Y 505.317,Z 1151.106,A -85,B 0,C 180,E1 24647.199,E2 24647.199} C_VEL
LIN {X 0,Y 506.171,Z 1141.573,A -85,B 0,C 180,E1 24645.005,E2 24645.005} C_VEL
LIN {X 0,Y 507.348,Z 1130.097,A -85,B 0,C 180,E1 24642.808,E2 24642.808} C_VEL
LIN {X 0,Y 508.81,Z 1117.213,A -85,B 0,C 180,E1 24640.725,E2 24640.725} C_VEL
LIN {X 0,Y 510.521,Z 1102.925,A -85,B 0,C 180,E1 24638.759,E2 24638.759} C_VEL
LIN {X 0,Y 512.451,Z 1087.046,A -85,B 0,C 180,E1 24636.912,E2 24636.912} C_VEL
LIN {X 0,Y 514.481,Z 1070.284,A -85,B 0,C 180,E1 24635.243,E2 24635.243} C_VEL
LIN {X 0,Y 516.631,Z 1052.088,A -85,B 0,C 180,E1 24633.695,E2 24633.695} C_VEL
LIN {X 0,Y 518.85,Z 1032.219,A -85,B 0,C 180,E1 24632.267,E2 24632.267} C_VEL
LIN {X 0,Y 520.879,Z 1012.13,A -85,B 0,C 180,E1 24631.073,E2 24631.073} C_VEL
LIN {X 0,Y 522.739,Z 991.357,A -85,B 0,C 180,E1 24630.054,E2 24630.054} C_VEL
LIN {X 0,Y 524.449,Z 969.455,A -85,B 0,C 180,E1 24629.192,E2 24629.192} C_VEL
LIN {X 0,Y 525.846,Z 947.127,A -85,B 0,C 180,E1 24628.518,E2 24628.518} C_VEL
LIN {X 0,Y 526.879,Z 924.049,A -85,B 0,C 180,E1 24628.034,E2 24628.034} C_VEL
LIN {X 0,Y 534.966,Z 697.836,A -85,B 0,C 180,E1 24624.329,E2 24624.329} C_VEL
LIN {X 0,Y 535.053,Z 690.724,A -85,B 0,C 180,E1 24624.199,E2 24624.199} C_VEL
LIN {X 0,Y 524.216,Z 670.729,A -85,B 0,C 180,E1 24623.055,E2 24623.055} C_VEL
LIN {X 0,Y 507.264,Z 641.283,A -85,B 0,C 180,E1 24621.179,E2 24621.179} C_VEL
LIN {X 0,Y 505.896,Z 637.826,A -85,B 0,C 180,E1 24620.998,E2 24620.998} C_VEL
LIN {X 0,Y 505.866,Z 637.656,A -85,B 0,C 180,E1 24617.473,E2 24617.473} C_VEL
LIN {X 0,Y 505.872,Z 637.654,A -85,B 0,C 180,E1 24613.931,E2 24613.931} C_VEL
LIN {X 0,Y 505.815,Z 637.662,A -85,B 0,C 180,E1 24610.57,E2 24610.57} C_VEL
LIN {X 0,Y 505.805,Z 637.66,A -85,B 0,C 180,E1 24607.081,E2 24607.081} C_VEL
LIN {X 0,Y 505.848,Z 637.656,A -85,B 0,C 180,E1 24603.606,E2 24603.606} C_VEL
LIN {X 0,Y 505.863,Z 637.652,A -85,B 0,C 180,E1 24600.137,E2 24600.137} C_VEL
LIN {X 0,Y 505.839,Z 637.655,A -85,B 0,C 180,E1 24596.662,E2 24596.662} C_VEL
LIN {X 0,Y 505.832,Z 637.658,A -85,B 0,C 180,E1 24593.203,E2 24593.203} C_VEL
LIN {X 0,Y 505.848,Z 637.661,A -85,B 0,C 180,E1 24589.757,E2 24589.757} C_VEL
LIN {X 0,Y 505.852,Z 637.654,A -85,B 0,C 180,E1 24587.336,E2 24587.336} C_VEL
LIN {X 0,Y 504.831,Z 637.782,A -85,B 0,C 180,E1 24586.464,E2 24586.464} C_VEL
LIN {X 0,Y 498.455,Z 638.571,A -85,B 0,C 180,E1 24584.011,E2 24584.011} C_VEL
LIN {X 0,Y 497.931,Z 638.632,A -85,B 0,C 180,E1 24583.372,E2 24583.372} C_VEL
LIN {X 0,Y 497.906,Z 638.641,A -85,B 0,C 180,E1 24579.83,E2 24579.83} C_VEL
LIN {X 0,Y 497.876,Z 638.65,A -85,B 0,C 180,E1 24576.227,E2 24576.227} C_VEL
LIN {X 0,Y 497.878,Z 638.637,A -85,B 0,C 180,E1 24572.764,E2 24572.764} C_VEL
LIN {X 0,Y 497.936,Z 638.645,A -85,B 0,C 180,E1 24569.311,E2 24569.311} C_VEL
LIN {X 0,Y 497.922,Z 638.631,A -85,B 0,C 180,E1 24565.741,E2 24565.741} C_VEL
LIN {X 0,Y 497.933,Z 638.646,A -85,B 0,C 180,E1 24562.153,E2 24562.153} C_VEL
LIN {X 0,Y 497.921,Z 638.627,A -85,B 0,C 180,E1 24558.652,E2 24558.652} C_VEL
LIN {X 0,Y 497.856,Z 638.65,A -85,B 0,C 180,E1 24555.224,E2 24555.224} C_VEL
LIN {X 0,Y 497.881,Z 638.646,A -85,B 0,C 180,E1 24551.744,E2 24551.744} C_VEL
LIN {X 0,Y 497.93,Z 638.641,A -85,B 0,C 180,E1 24548.318,E2 24548.318} C_VEL
LIN {X 0,Y 497.914,Z 638.643,A -85,B 0,C 180,E1 24544.805,E2 24544.805} C_VEL
LIN {X 0,Y 497.89,Z 638.649,A -85,B 0,C 180,E1 24541.319,E2 24541.319} C_VEL
LIN {X 0,Y 497.901,Z 638.649,A -85,B 0,C 180,E1 24537.93,E2 24537.93} C_VEL
LIN {X 0,Y 497.913,Z 638.648,A -85,B 0,C 180,E1 24534.385,E2 24534.385} C_VEL
LIN {X 0,Y 497.912,Z 638.648,A -85,B 0,C 180,E1 24530.911,E2 24530.911} C_VEL
LIN {X 0,Y 497.928,Z 638.643,A -85,B 0,C 180,E1 24527.414,E2 24527.414} C_VEL
LIN {X 0,Y 497.946,Z 638.761,A -85,B 0,C 180,E1 24525.269,E2 24525.269} C_VEL
LIN {X 0,Y 506.081,Z 666.742,A -85,B 0,C 180,E1 24522.447,E2 24522.447} C_VEL
LIN {X 0,Y 508.955,Z 677.624,A -85,B 0,C 180,E1 24521.372,E2 24521.372} C_VEL
LIN {X 0,Y 507.474,Z 721.006,A -85,B 0,C 180,E1 24517.786,E2 24517.786} C_VEL
LIN {X 0,Y 506.001,Z 763.234,A -85,B 0,C 180,E1 24514.315,E2 24514.315} C_VEL
LIN {X 0,Y 504.597,Z 805.106,A -85,B 0,C 180,E1 24510.875,E2 24510.875} C_VEL
LIN {X 0,Y 503.656,Z 836.481,A -85,B 0,C 180,E1 24508.345,E2 24508.345} C_VEL
LIN {X 0,Y 502.962,Z 884.157,A -85,B 0,C 180,E1 24507.526,E2 24507.526} C_VEL
LIN {X 0,Y 501.577,Z 979.419,A -85,B 0,C 180,E1 24505.91,E2 24505.91} C_VEL
LIN {X 0,Y 501.392,Z 995.41,A -85,B 0,C 180,E1 24505.449,E2 24505.449} C_VEL
LIN {X 0,Y 501.005,Z 1011.688,A -85,B 0,C 180,E1 24504.765,E2 24504.765} C_VEL
LIN {X 0,Y 500.531,Z 1026.585,A -85,B 0,C 180,E1 24503.921,E2 24503.921} C_VEL
LIN {X 0,Y 499.943,Z 1041.593,A -85,B 0,C 180,E1 24502.827,E2 24502.827} C_VEL
LIN {X 0,Y 499.307,Z 1055.221,A -85,B 0,C 180,E1 24501.556,E2 24501.556} C_VEL
LIN {X 0,Y 498.753,Z 1066.532,A -85,B 0,C 180,E1 24500.25,E2 24500.25} C_VEL
LIN {X 0,Y 498.202,Z 1077.293,A -85,B 0,C 180,E1 24498.691,E2 24498.691} C_VEL
LIN {X 0,Y 497.811,Z 1085.645,A -85,B 0,C 180,E1 24497.17,E2 24497.17} C_VEL
LIN {X 0,Y 497.503,Z 1093.179,A -85,B 0,C 180,E1 24495.382,E2 24495.382} C_VEL
LIN {X 0,Y 497.333,Z 1098.299,A -85,B 0,C 180,E1 24493.721,E2 24493.721} C_VEL
LIN {X 0,Y 497.259,Z 1102.133,A -85,B 0,C 180,E1 24491.833,E2 24491.833} C_VEL
LIN {X 0,Y 497.309,Z 1103.941,A -85,B 0,C 180,E1 24490.071,E2 24490.071} C_VEL
LIN {X 0,Y 497.462,Z 1103.996,A -85,B 0,C 180,E1 24488.202,E2 24488.202} C_VEL
LIN {X 0,Y 497.729,Z 1102.345,A -85,B 0,C 180,E1 24486.457,E2 24486.457} C_VEL
LIN {X 0,Y 498.151,Z 1098.665,A -85,B 0,C 180,E1 24484.603,E2 24484.603} C_VEL
LIN {X 0,Y 498.696,Z 1093.384,A -85,B 0,C 180,E1 24482.871,E2 24482.871} C_VEL
LIN {X 0,Y 499.406,Z 1086.045,A -85,B 0,C 180,E1 24481.145,E2 24481.145} C_VEL
LIN {X 0,Y 500.185,Z 1077.792,A -85,B 0,C 180,E1 24479.654,E2 24479.654} C_VEL
LIN {X 0,Y 501.093,Z 1067.309,A -85,B 0,C 180,E1 24478.168,E2 24478.168} C_VEL
LIN {X 0,Y 501.993,Z 1055.697,A -85,B 0,C 180,E1 24476.858,E2 24476.858} C_VEL
LIN {X 0,Y 502.916,Z 1041.747,A -85,B 0,C 180,E1 24475.608,E2 24475.608} C_VEL
LIN {X 0,Y 503.621,Z 1027.988,A -85,B 0,C 180,E1 24474.643,E2 24474.643} C_VEL
LIN {X 0,Y 504.165,Z 1014.375,A -85,B 0,C 180,E1 24473.907,E2 24473.907} C_VEL
LIN {X 0,Y 504.54,Z 1001.799,A -85,B 0,C 180,E1 24473.376,E2 24473.376} C_VEL
LIN {X 0,Y 504.791,Z 987.089,A -85,B 0,C 180,E1 24472.912,E2 24472.912} C_VEL
LIN {X 0,Y 505.356,Z 946.094,A -85,B 0,C 180,E1 24472.14,E2 24472.14} C_VEL
LIN {X 0,Y 508.439,Z 845.558,A -85,B 0,C 180,E1 24470.261,E2 24470.261} C_VEL
LIN {X 0,Y 508.926,Z 841.178,A -85,B 0,C 180,E1 24469.927,E2 24469.927} C_VEL
LIN {X 0,Y 510.756,Z 797.317,A -85,B 0,C 180,E1 24466.353,E2 24466.353} C_VEL
LIN {X 0,Y 512.447,Z 753.906,A -85,B 0,C 180,E1 24462.862,E2 24462.862} C_VEL
LIN {X 0,Y 514.065,Z 713.226,A -85,B 0,C 180,E1 24459.623,E2 24459.623} C_VEL
LIN {X 0,Y 515.202,Z 682.553,A -85,B 0,C 180,E1 24457.194,E2 24457.194} C_VEL
LIN {X 0,Y 510.959,Z 668.561,A -85,B 0,C 180,E1 24455.611,E2 24455.611} C_VEL
LIN {X 0,Y 505.412,Z 654.568,A -85,B 0,C 180,E1 24453.819,E2 24453.819} C_VEL
LIN {X 0,Y 501.502,Z 646.495,A -85,B 0,C 180,E1 24452.647,E2 24452.647} C_VEL
LIN {X 0,Y 499.667,Z 642.738,A -85,B 0,C 180,E1 24452.076,E2 24452.076} C_VEL
LIN {X 0,Y 498.045,Z 639.344,A -85,B 0,C 180,E1 24451.558,E2 24451.558} C_VEL
LIN {X 0,Y 497.917,Z 638.647,A -85,B 0,C 180,E1 24451.447,E2 24451.447} C_VEL
LIN {X 0,Y 497.907,Z 638.647,A -85,B 0,C 180,E1 24448.117,E2 24448.117} C_VEL
LIN {X 0,Y 497.924,Z 638.645,A -85,B 0,C 180,E1 24444.613,E2 24444.613} C_VEL
LIN {X 0,Y 497.928,Z 638.645,A -85,B 0,C 180,E1 24440.813,E2 24440.813} C_VEL
LIN {X 0,Y 497.931,Z 638.642,A -85,B 0,C 180,E1 24437.253,E2 24437.253} C_VEL
LIN {X 0,Y 497.916,Z 638.784,A -85,B 0,C 180,E1 24434.17,E2 24434.17} C_VEL
LIN {X 0,Y 505.33,Z 660.855,A -85,B 0,C 180,E1 24430.913,E2 24430.913} C_VEL
LIN {X 0,Y 510.426,Z 676.538,A -85,B 0,C 180,E1 24428.746,E2 24428.746} C_VEL
LIN {X 0,Y 523.259,Z 702.656,A -85,B 0,C 180,E1 24427.274,E2 24427.274} C_VEL
LIN {X 0,Y 528.241,Z 730.522,A -85,B 0,C 180,E1 24426.372,E2 24426.372} C_VEL
LIN {X 0,Y 519.764,Z 955.794,A -85,B 0,C 180,E1 24422.595,E2 24422.595} C_VEL
LIN {X 0,Y 518.433,Z 987.281,A -85,B 0,C 180,E1 24422.013,E2 24422.013} C_VEL
LIN {X 0,Y 516.908,Z 1010.01,A -85,B 0,C 180,E1 24421.398,E2 24421.398} C_VEL
LIN {X 0,Y 515.125,Z 1031.683,A -85,B 0,C 180,E1 24420.614,E2 24420.614} C_VEL
LIN {X 0,Y 513.067,Z 1052.949,A -85,B 0,C 180,E1 24419.633,E2 24419.633} C_VEL
LIN {X 0,Y 510.875,Z 1073.68,A -85,B 0,C 180,E1 24418.46,E2 24418.46} C_VEL
LIN {X 0,Y 508.631,Z 1093.28,A -85,B 0,C 180,E1 24417.132,E2 24417.132} C_VEL
LIN {X 0,Y 506.394,Z 1112.09,A -85,B 0,C 180,E1 24415.619,E2 24415.619} C_VEL
LIN {X 0,Y 504.26,Z 1129.301,A -85,B 0,C 180,E1 24413.983,E2 24413.983} C_VEL
LIN {X 0,Y 502.203,Z 1146.188,A -85,B 0,C 180,E1 24412.103,E2 24412.103} C_VEL
LIN {X 0,Y 500.511,Z 1160.721,A -85,B 0,C 180,E1 24410.217,E2 24410.217} C_VEL
LIN {X 0,Y 499.06,Z 1173.888,A -85,B 0,C 180,E1 24408.211,E2 24408.211} C_VEL
LIN {X 0,Y 497.903,Z 1185.737,A -85,B 0,C 180,E1 24406.087,E2 24406.087} C_VEL
LIN {X 0,Y 497.039,Z 1196.285,A -85,B 0,C 180,E1 24403.849,E2 24403.849} C_VEL
LIN {X 0,Y 496.475,Z 1204.927,A -85,B 0,C 180,E1 24401.617,E2 24401.617} C_VEL
LIN {X 0,Y 496.161,Z 1212.179,A -85,B 0,C 180,E1 24399.276,E2 24399.276} C_VEL
LIN {X 0,Y 496.025,Z 1217.77,A -85,B 0,C 180,E1 24396.945,E2 24396.945} C_VEL
LIN {X 0,Y 496.008,Z 1221.631,A -85,B 0,C 180,E1 24394.623,E2 24394.623} C_VEL
LIN {X 0,Y 496.039,Z 1224.019,A -85,B 0,C 180,E1 24392.193,E2 24392.193} C_VEL
LIN {X 0,Y 496.048,Z 1224.76,A -85,B 0,C 180,E1 24389.883,E2 24389.883} C_VEL
LIN {X 0,Y 496.038,Z 1223.845,A -85,B 0,C 180,E1 24387.572,E2 24387.572} C_VEL
LIN {X 0,Y 496.004,Z 1221.301,A -85,B 0,C 180,E1 24385.142,E2 24385.142} C_VEL
LIN {X 0,Y 496.042,Z 1217.23,A -85,B 0,C 180,E1 24382.819,E2 24382.819} C_VEL
LIN {X 0,Y 496.177,Z 1211.495,A -85,B 0,C 180,E1 24380.487,E2 24380.487} C_VEL
LIN {X 0,Y 496.521,Z 1204.104,A -85,B 0,C 180,E1 24378.145,E2 24378.145} C_VEL
LIN {X 0,Y 497.148,Z 1194.732,A -85,B 0,C 180,E1 24375.795,E2 24375.795} C_VEL
LIN {X 0,Y 498.071,Z 1183.926,A -85,B 0,C 180,E1 24373.556,E2 24373.556} C_VEL
LIN {X 0,Y 499.291,Z 1171.835,A -85,B 0,C 180,E1 24371.432,E2 24371.432} C_VEL
LIN {X 0,Y 500.809,Z 1158.355,A -85,B 0,C 180,E1 24369.426,E2 24369.426} C_VEL
LIN {X 0,Y 502.718,Z 1142.626,A -85,B 0,C 180,E1 24367.425,E2 24367.425} C_VEL
LIN {X 0,Y 504.986,Z 1124.785,A -85,B 0,C 180,E1 24365.491,E2 24365.491} C_VEL
LIN {X 0,Y 507.345,Z 1106.511,A -85,B 0,C 180,E1 24363.801,E2 24363.801} C_VEL
LIN {X 0,Y 509.901,Z 1086.607,A -85,B 0,C 180,E1 24362.242,E2 24362.242} C_VEL
LIN {X 0,Y 512.472,Z 1065.745,A -85,B 0,C 180,E1 24360.868,E2 24360.868} C_VEL
LIN {X 0,Y 515.038,Z 1044.158,A -85,B 0,C 180,E1 24359.683,E2 24359.683} C_VEL
LIN {X 0,Y 517.62,Z 1020.713,A -85,B 0,C 180,E1 24358.632,E2 24358.632} C_VEL
LIN {X 0,Y 520.034,Z 997.222,A -85,B 0,C 180,E1 24357.804,E2 24357.804} C_VEL
LIN {X 0,Y 522.14,Z 973.189,A -85,B 0,C 180,E1 24357.16,E2 24357.16} C_VEL
LIN {X 0,Y 528.455,Z 880.056,A -85,B 0,C 180,E1 24355.197,E2 24355.197} C_VEL
LIN {X 0,Y 535.683,Z 800.549,A -85,B 0,C 180,E1 24353.397,E2 24353.397} C_VEL
LIN {X 0,Y 543.44,Z 731.968,A -85,B 0,C 180,E1 24351.761,E2 24351.761} C_VEL
LIN {X 0,Y 543.113,Z 715.183,A -85,B 0,C 180,E1 24350.877,E2 24350.877} C_VEL
LIN {X 0,Y 540.558,Z 707.597,A -85,B 0,C 180,E1 24349.883,E2 24349.883} C_VEL
LIN {X 0,Y 538.727,Z 702.663,A -85,B 0,C 180,E1 24349.063,E2 24349.063} C_VEL
LIN {X 0,Y 536.391,Z 696.582,A -85,B 0,C 180,E1 24347.738,E2 24347.738} C_VEL
LIN {X 0,Y 534.655,Z 692.236,A -85,B 0,C 180,E1 24346.212,E2 24346.212} C_VEL
LIN {X 0,Y 534.199,Z 689.662,A -85,B 0,C 180,E1 24344.582,E2 24344.582} C_VEL
LIN {X 0,Y 535.135,Z 689.802,A -85,B 0,C 180,E1 24342.856,E2 24342.856} C_VEL
LIN {X 0,Y 536.41,Z 690.966,A -85,B 0,C 180,E1 24341.863,E2 24341.863} C_VEL
LIN {X 0,Y 538.737,Z 694.328,A -85,B 0,C 180,E1 24340.569,E2 24340.569} C_VEL
LIN {X 0,Y 540.454,Z 696.863,A -85,B 0,C 180,E1 24339.843,E2 24339.843} C_VEL
LIN {X 0,Y 543.607,Z 702.104,A -85,B 0,C 180,E1 24338.725,E2 24338.725} C_VEL
LIN {X 0,Y 545.839,Z 706.655,A -85,B 0,C 180,E1 24338.02,E2 24338.02} C_VEL
LIN {X 0,Y 536.218,Z 785.672,A -85,B 0,C 180,E1 24336.137,E2 24336.137} C_VEL
LIN {X 0,Y 528.886,Z 862.97,A -85,B 0,C 180,E1 24334.378,E2 24334.378} C_VEL
LIN {X 0,Y 522.966,Z 946.159,A -85,B 0,C 180,E1 24332.572,E2 24332.572} C_VEL
LIN {X 0,Y 521.191,Z 968.911,A -85,B 0,C 180,E1 24331.876,E2 24331.876} C_VEL
LIN {X 0,Y 519.116,Z 990.966,A -85,B 0,C 180,E1 24331.003,E2 24331.003} C_VEL
LIN {X 0,Y 516.813,Z 1012.29,A -85,B 0,C 180,E1 24329.946,E2 24329.946} C_VEL
LIN {X 0,Y 514.461,Z 1031.941,A -85,B 0,C 180,E1 24328.77,E2 24328.77} C_VEL
LIN {X 0,Y 511.938,Z 1051.519,A -85,B 0,C 180,E1 24327.374,E2 24327.374} C_VEL
LIN {X 0,Y 509.445,Z 1069.809,A -85,B 0,C 180,E1 24325.833,E2 24325.833} C_VEL
LIN {X 0,Y 506.935,Z 1087.179,A -85,B 0,C 180,E1 24324.1,E2 24324.1} C_VEL
LIN {X 0,Y 504.612,Z 1102.985,A -85,B 0,C 180,E1 24322.241,E2 24322.241} C_VEL
LIN {X 0,Y 502.405,Z 1118.138,A -85,B 0,C 180,E1 24320.142,E2 24320.142} C_VEL
LIN {X 0,Y 500.611,Z 1130.982,A -85,B 0,C 180,E1 24318.037,E2 24318.037} C_VEL
LIN {X 0,Y 499.189,Z 1141.811,A -85,B 0,C 180,E1 24315.929,E2 24315.929} C_VEL
LIN {X 0,Y 498.026,Z 1151.515,A -85,B 0,C 180,E1 24313.654,E2 24313.654} C_VEL
LIN {X 0,Y 497.156,Z 1159.866,A -85,B 0,C 180,E1 24311.252,E2 24311.252} C_VEL
LIN {X 0,Y 496.622,Z 1166.269,A -85,B 0,C 180,E1 24308.921,E2 24308.921} C_VEL
LIN {X 0,Y 496.305,Z 1170.943,A -85,B 0,C 180,E1 24306.597,E2 24306.597} C_VEL
LIN {X 0,Y 496.127,Z 1174.399,A -85,B 0,C 180,E1 24304.047,E2 24304.047} C_VEL
LIN {X 0,Y 496.073,Z 1176.091,A -85,B 0,C 180,E1 24301.619,E2 24301.619} C_VEL
LIN {X 0,Y 496.055,Z 1176.057,A -85,B 0,C 180,E1 24299.194,E2 24299.194} C_VEL
LIN {X 0,Y 496.07,Z 1174.362,A -85,B 0,C 180,E1 24296.652,E2 24296.652} C_VEL
LIN {X 0,Y 496.152,Z 1171.135,A -85,B 0,C 180,E1 24294.219,E2 24294.219} C_VEL
LIN {X 0,Y 496.34,Z 1166.393,A -85,B 0,C 180,E1 24291.896,E2 24291.896} C_VEL
LIN {X 0,Y 496.738,Z 1159.714,A -85,B 0,C 180,E1 24289.448,E2 24289.448} C_VEL
LIN {X 0,Y 497.368,Z 1151.614,A -85,B 0,C 180,E1 24287.109,E2 24287.109} C_VEL
LIN {X 0,Y 498.308,Z 1141.531,A -85,B 0,C 180,E1 24284.763,E2 24284.763} C_VEL
LIN {X 0,Y 499.55,Z 1129.926,A -85,B 0,C 180,E1 24282.531,E2 24282.531} C_VEL
LIN {X 0,Y 501.178,Z 1116.1,A -85,B 0,C 180,E1 24280.299,E2 24280.299} C_VEL
LIN {X 0,Y 502.996,Z 1101.51,A -85,B 0,C 180,E1 24278.303,E2 24278.303} C_VEL
LIN {X 0,Y 505.033,Z 1085.418,A -85,B 0,C 180,E1 24276.429,E2 24276.429} C_VEL
LIN {X 0,Y 507.177,Z 1068.23,A -85,B 0,C 180,E1 24274.737,E2 24274.737} C_VEL
LIN {X 0,Y 509.421,Z 1049.511,A -85,B 0,C 180,E1 24273.167,E2 24273.167} C_VEL
LIN {X 0,Y 511.649,Z 1029.91,A -85,B 0,C 180,E1 24271.779,E2 24271.779} C_VEL
LIN {X 0,Y 513.779,Z 1009.49,A -85,B 0,C 180,E1 24270.571,E2 24270.571} C_VEL
LIN {X 0,Y 515.729,Z 987.947,A -85,B 0,C 180,E1 24269.54,E2 24269.54} C_VEL
LIN {X 0,Y 517.407,Z 966.034,A -85,B 0,C 180,E1 24268.706,E2 24268.706} C_VEL
LIN {X 0,Y 518.784,Z 943.354,A -85,B 0,C 180,E1 24268.049,E2 24268.049} C_VEL
LIN {X 0,Y 519.838,Z 920.274,A -85,B 0,C 180,E1 24267.582,E2 24267.582} C_VEL
LIN {X 0,Y 527.628,Z 710.689,A -85,B 0,C 180,E1 24264.09,E2 24264.09} C_VEL
LIN {X 0,Y 528.209,Z 693.512,A -85,B 0,C 180,E1 24263.789,E2 24263.789} C_VEL
LIN {X 0,Y 516.904,Z 672.66,A -85,B 0,C 180,E1 24262.568,E2 24262.568} C_VEL
LIN {X 0,Y 499.284,Z 642.185,A -85,B 0,C 180,E1 24260.582,E2 24260.582} C_VEL
LIN {X 0,Y 497.942,Z 638.707,A -85,B 0,C 180,E1 24260.398,E2 24260.398} C_VEL
LIN {X 0,Y 497.916,Z 638.645,A -85,B 0,C 180,E1 24256.944,E2 24256.944} C_VEL
LIN {X 0,Y 497.896,Z 638.65,A -85,B 0,C 180,E1 24253.371,E2 24253.371} C_VEL
LIN {X 0,Y 497.9,Z 638.646,A -85,B 0,C 180,E1 24249.908,E2 24249.908} C_VEL
LIN {X 0,Y 497.912,Z 638.649,A -85,B 0,C 180,E1 24246.369,E2 24246.369} C_VEL
LIN {X 0,Y 497.916,Z 638.644,A -85,B 0,C 180,E1 24242.835,E2 24242.835} C_VEL
LIN {X 0,Y 497.929,Z 638.641,A -85,B 0,C 180,E1 24239.34,E2 24239.34} C_VEL
LIN {X 0,Y 497.918,Z 638.64,A -85,B 0,C 180,E1 24235.835,E2 24235.835} C_VEL
LIN {X 0,Y 497.854,Z 638.647,A -85,B 0,C 180,E1 24232.434,E2 24232.434} C_VEL
LIN {X 0,Y 497.872,Z 638.646,A -85,B 0,C 180,E1 24228.866,E2 24228.866} C_VEL
LIN {X 0,Y 497.933,Z 638.641,A -85,B 0,C 180,E1 24225.461,E2 24225.461} C_VEL
LIN {X 0,Y 497.931,Z 638.632,A -85,B 0,C 180,E1 24223.372,E2 24223.372} C_VEL
LIN {X 0,Y 496.935,Z 638.763,A -85,B 0,C 180,E1 24222.486,E2 24222.486} C_VEL
LIN {X 0,Y 490.495,Z 639.567,A -85,B 0,C 180,E1 24219.994,E2 24219.994} C_VEL
LIN {X 0,Y 489.985,Z 639.628,A -85,B 0,C 180,E1 24219.344,E2 24219.344} C_VEL
LIN {X 0,Y 489.932,Z 639.638,A -85,B 0,C 180,E1 24215.976,E2 24215.976} C_VEL
LIN {X 0,Y 489.916,Z 639.628,A -85,B 0,C 180,E1 24212.341,E2 24212.341} C_VEL
LIN {X 0,Y 489.985,Z 639.631,A -85,B 0,C 180,E1 24208.949,E2 24208.949} C_VEL
LIN {X 0,Y 489.987,Z 639.621,A -85,B 0,C 180,E1 24205.437,E2 24205.437} C_VEL
LIN {X 0,Y 489.981,Z 639.634,A -85,B 0,C 180,E1 24201.907,E2 24201.907} C_VEL
LIN {X 0,Y 489.975,Z 639.618,A -85,B 0,C 180,E1 24198.346,E2 24198.346} C_VEL
LIN {X 0,Y 489.964,Z 639.639,A -85,B 0,C 180,E1 24194.739,E2 24194.739} C_VEL
LIN {X 0,Y 489.964,Z 639.637,A -85,B 0,C 180,E1 24191.192,E2 24191.192} C_VEL
LIN {X 0,Y 489.976,Z 639.634,A -85,B 0,C 180,E1 24187.695,E2 24187.695} C_VEL
LIN {X 0,Y 489.995,Z 639.63,A -85,B 0,C 180,E1 24184.109,E2 24184.109} C_VEL
LIN {X 0,Y 489.946,Z 639.637,A -85,B 0,C 180,E1 24180.675,E2 24180.675} C_VEL
LIN {X 0,Y 489.915,Z 639.641,A -85,B 0,C 180,E1 24177.122,E2 24177.122} C_VEL
LIN {X 0,Y 489.956,Z 639.635,A -85,B 0,C 180,E1 24173.571,E2 24173.571} C_VEL
LIN {X 0,Y 489.998,Z 639.632,A -85,B 0,C 180,E1 24170.104,E2 24170.104} C_VEL
LIN {X 0,Y 489.972,Z 639.631,A -85,B 0,C 180,E1 24166.553,E2 24166.553} C_VEL
LIN {X 0,Y 490.003,Z 639.69,A -85,B 0,C 180,E1 24165.648,E2 24165.648} C_VEL
LIN {X 0,Y 498.108,Z 667.321,A -85,B 0,C 180,E1 24162.806,E2 24162.806} C_VEL
LIN {X 0,Y 501.395,Z 680.369,A -85,B 0,C 180,E1 24161.531,E2 24161.531} C_VEL
LIN {X 0,Y 499.863,Z 723.209,A -85,B 0,C 180,E1 24157.962,E2 24157.962} C_VEL
LIN {X 0,Y 498.353,Z 764.589,A -85,B 0,C 180,E1 24154.535,E2 24154.535} C_VEL
LIN {X 0,Y 496.896,Z 806.057,A -85,B 0,C 180,E1 24151.099,E2 24151.099} C_VEL
LIN {X 0,Y 495.937,Z 837.254,A -85,B 0,C 180,E1 24148.572,E2 24148.572} C_VEL
LIN {X 0,Y 493.727,Z 981.235,A -85,B 0,C 180,E1 24146.055,E2 24146.055} C_VEL
LIN {X 0,Y 493.501,Z 998.111,A -85,B 0,C 180,E1 24145.539,E2 24145.539} C_VEL
LIN {X 0,Y 493.11,Z 1013.603,A -85,B 0,C 180,E1 24144.862,E2 24144.862} C_VEL
LIN {X 0,Y 492.596,Z 1029.065,A -85,B 0,C 180,E1 24143.948,E2 24143.948} C_VEL
LIN {X 0,Y 492.021,Z 1043.03,A -85,B 0,C 180,E1 24142.897,E2 24142.897} C_VEL
LIN {X 0,Y 491.362,Z 1056.871,A -85,B 0,C 180,E1 24141.577,E2 24141.577} C_VEL
LIN {X 0,Y 490.797,Z 1067.949,A -85,B 0,C 180,E1 24140.26,E2 24140.26} C_VEL
LIN {X 0,Y 490.241,Z 1078.686,A -85,B 0,C 180,E1 24138.673,E2 24138.673} C_VEL
LIN {X 0,Y 489.836,Z 1087.097,A -85,B 0,C 180,E1 24137.091,E2 24137.091} C_VEL
LIN {X 0,Y 489.55,Z 1094.111,A -85,B 0,C 180,E1 24135.395,E2 24135.395} C_VEL
LIN {X 0,Y 489.377,Z 1099.253,A -85,B 0,C 180,E1 24133.707,E2 24133.707} C_VEL
LIN {X 0,Y 489.31,Z 1103.11,A -85,B 0,C 180,E1 24131.788,E2 24131.788} C_VEL
LIN {X 0,Y 489.37,Z 1104.927,A -85,B 0,C 180,E1 24129.999,E2 24129.999} C_VEL
LIN {X 0,Y 489.541,Z 1104.994,A -85,B 0,C 180,E1 24128.099,E2 24128.099} C_VEL
LIN {X 0,Y 489.848,Z 1103.255,A -85,B 0,C 180,E1 24126.264,E2 24126.264} C_VEL
LIN {X 0,Y 490.331,Z 1099.397,A -85,B 0,C 180,E1 24124.324,E2 24124.324} C_VEL
LIN {X 0,Y 490.927,Z 1093.946,A -85,B 0,C 180,E1 24122.566,E2 24122.566} C_VEL
LIN {X 0,Y 491.712,Z 1086.47,A -85,B 0,C 180,E1 24120.813,E2 24120.813} C_VEL
LIN {X 0,Y 492.548,Z 1077.985,A -85,B 0,C 180,E1 24119.3,E2 24119.3} C_VEL
LIN {X 0,Y 493.537,Z 1067.362,A -85,B 0,C 180,E1 24117.791,E2 24117.791} C_VEL
LIN {X 0,Y 494.505,Z 1055.494,A -85,B 0,C 180,E1 24116.462,E2 24116.462} C_VEL
LIN {X 0,Y 495.4,Z 1042.675,A -85,B 0,C 180,E1 24115.309,E2 24115.309} C_VEL
LIN {X 0,Y 496.194,Z 1027.926,A -85,B 0,C 180,E1 24114.273,E2 24114.273} C_VEL
LIN {X 0,Y 496.72,Z 1015.146,A -85,B 0,C 180,E1 24113.583,E2 24113.583} C_VEL
LIN {X 0,Y 497.11,Z 1002.676,A -85,B 0,C 180,E1 24113.052,E2 24113.052} C_VEL
LIN {X 0,Y 497.373,Z 987.992,A -85,B 0,C 180,E1 24112.584,E2 24112.584} C_VEL
LIN {X 0,Y 497.958,Z 948.762,A -85,B 0,C 180,E1 24111.819,E2 24111.819} C_VEL
LIN {X 0,Y 501.312,Z 846.744,A -85,B 0,C 180,E1 24109.86,E2 24109.86} C_VEL
LIN {X 0,Y 501.837,Z 842.05,A -85,B 0,C 180,E1 24109.493,E2 24109.493} C_VEL
LIN {X 0,Y 503.559,Z 802.013,A -85,B 0,C 180,E1 24106.213,E2 24106.213} C_VEL
LIN {X 0,Y 505.371,Z 760.717,A -85,B 0,C 180,E1 24102.852,E2 24102.852} C_VEL
LIN {X 0,Y 507.101,Z 721.567,A -85,B 0,C 180,E1 24099.692,E2 24099.692} C_VEL
LIN {X 0,Y 508.693,Z 686.109,A -85,B 0,C 180,E1 24096.849,E2 24096.849} C_VEL
LIN {X 0,Y 504.654,Z 672.647,A -85,B 0,C 180,E1 24095.286,E2 24095.286} C_VEL
LIN {X 0,Y 499.264,Z 658.966,A -85,B 0,C 180,E1 24093.472,E2 24093.472} C_VEL
LIN {X 0,Y 494.266,Z 648.411,A -85,B 0,C 180,E1 24091.876,E2 24091.876} C_VEL
LIN {X 0,Y 491.994,Z 644.046,A -85,B 0,C 180,E1 24091.15,E2 24091.15} C_VEL
LIN {X 0,Y 490.176,Z 640.721,A -85,B 0,C 180,E1 24090.572,E2 24090.572} C_VEL
LIN {X 0,Y 489.974,Z 639.635,A -85,B 0,C 180,E1 24090.404,E2 24090.404} C_VEL
LIN {X 0,Y 489.959,Z 639.638,A -85,B 0,C 180,E1 24086.981,E2 24086.981} C_VEL
LIN {X 0,Y 489.985,Z 639.632,A -85,B 0,C 180,E1 24083.511,E2 24083.511} C_VEL
LIN {X 0,Y 489.974,Z 639.634,A -85,B 0,C 180,E1 24080.109,E2 24080.109} C_VEL
LIN {X 0,Y 489.985,Z 639.628,A -85,B 0,C 180,E1 24076.388,E2 24076.388} C_VEL
LIN {X 0,Y 489.98,Z 639.689,A -85,B 0,C 180,E1 24074.748,E2 24074.748} C_VEL
LIN {X 0,Y 497.457,Z 661.993,A -85,B 0,C 180,E1 24071.395,E2 24071.395} C_VEL
LIN {X 0,Y 502.155,Z 676.31,A -85,B 0,C 180,E1 24069.389,E2 24069.389} C_VEL
LIN {X 0,Y 516.782,Z 705.854,A -85,B 0,C 180,E1 24067.663,E2 24067.663} C_VEL
LIN {X 0,Y 521.388,Z 731.922,A -85,B 0,C 180,E1 24066.81,E2 24066.81} C_VEL
LIN {X 0,Y 512.37,Z 961.566,A -85,B 0,C 180,E1 24062.888,E2 24062.888} C_VEL
LIN {X 0,Y 511.137,Z 988.057,A -85,B 0,C 180,E1 24062.372,E2 24062.372} C_VEL
LIN {X 0,Y 509.499,Z 1011.237,A -85,B 0,C 180,E1 24061.721,E2 24061.721} C_VEL
LIN {X 0,Y 507.677,Z 1032.536,A -85,B 0,C 180,E1 24060.932,E2 24060.932} C_VEL
LIN {X 0,Y 505.484,Z 1054.363,A -85,B 0,C 180,E1 24059.897,E2 24059.897} C_VEL
LIN {X 0,Y 503.28,Z 1074.325,A -85,B 0,C 180,E1 24058.735,E2 24058.735} C_VEL
LIN {X 0,Y 500.875,Z 1094.508,A -85,B 0,C 180,E1 24057.33,E2 24057.33} C_VEL
LIN {X 0,Y 498.586,Z 1113.117,A -85,B 0,C 180,E1 24055.795,E2 24055.795} C_VEL
LIN {X 0,Y 496.331,Z 1130.744,A -85,B 0,C 180,E1 24054.074,E2 24054.074} C_VEL
LIN {X 0,Y 494.296,Z 1146.884,A -85,B 0,C 180,E1 24052.225,E2 24052.225} C_VEL
LIN {X 0,Y 492.469,Z 1162.087,A -85,B 0,C 180,E1 24050.19,E2 24050.19} C_VEL
LIN {X 0,Y 491.012,Z 1175.123,A -85,B 0,C 180,E1 24048.152,E2 24048.152} C_VEL
LIN {X 0,Y 489.833,Z 1186.903,A -85,B 0,C 180,E1 24045.957,E2 24045.957} C_VEL
LIN {X 0,Y 488.957,Z 1197.491,A -85,B 0,C 180,E1 24043.6,E2 24043.6} C_VEL
LIN {X 0,Y 488.42,Z 1206.021,A -85,B 0,C 180,E1 24041.296,E2 24041.296} C_VEL
LIN {X 0,Y 488.138,Z 1212.863,A -85,B 0,C 180,E1 24038.954,E2 24038.954} C_VEL
LIN {X 0,Y 488.024,Z 1218.114,A -85,B 0,C 180,E1 24036.587,E2 24036.587} C_VEL
LIN {X 0,Y 488.026,Z 1221.804,A -85,B 0,C 180,E1 24034.228,E2 24034.228} C_VEL
LIN {X 0,Y 488.052,Z 1223.782,A -85,B 0,C 180,E1 24031.877,E2 24031.877} C_VEL
LIN {X 0,Y 488.051,Z 1224.272,A -85,B 0,C 180,E1 24029.411,E2 24029.411} C_VEL
LIN {X 0,Y 488.031,Z 1223.206,A -85,B 0,C 180,E1 24027.18,E2 24027.18} C_VEL
LIN {X 0,Y 488.009,Z 1220.389,A -85,B 0,C 180,E1 24024.708,E2 24024.708} C_VEL
LIN {X 0,Y 488.05,Z 1216.149,A -85,B 0,C 180,E1 24022.346,E2 24022.346} C_VEL
LIN {X 0,Y 488.231,Z 1210.122,A -85,B 0,C 180,E1 24019.973,E2 24019.973} C_VEL
LIN {X 0,Y 488.679,Z 1201.799,A -85,B 0,C 180,E1 24017.426,E2 24017.426} C_VEL
LIN {X 0,Y 489.407,Z 1192.287,A -85,B 0,C 180,E1 24015.081,E2 24015.081} C_VEL
LIN {X 0,Y 490.478,Z 1181.068,A -85,B 0,C 180,E1 24012.805,E2 24012.805} C_VEL
LIN {X 0,Y 491.906,Z 1168.112,A -85,B 0,C 180,E1 24010.594,E2 24010.594} C_VEL
LIN {X 0,Y 493.69,Z 1153.663,A -85,B 0,C 180,E1 24008.493,E2 24008.493} C_VEL
LIN {X 0,Y 495.782,Z 1137.842,A -85,B 0,C 180,E1 24006.526,E2 24006.526} C_VEL
LIN {X 0,Y 498.121,Z 1120.429,A -85,B 0,C 180,E1 24004.686,E2 24004.686} C_VEL
LIN {X 0,Y 500.726,Z 1101.505,A -85,B 0,C 180,E1 24002.979,E2 24002.979} C_VEL
LIN {X 0,Y 503.5,Z 1080.931,A -85,B 0,C 180,E1 24001.405,E2 24001.405} C_VEL
LIN {X 0,Y 506.214,Z 1060.409,A -85,B 0,C 180,E1 24000.082,E2 24000.082} C_VEL
LIN {X 0,Y 509.005,Z 1038.168,A -85,B 0,C 180,E1 23998.892,E2 23998.892} C_VEL
LIN {X 0,Y 511.694,Z 1015.019,A -85,B 0,C 180,E1 23997.891,E2 23997.891} C_VEL
LIN {X 0,Y 514.217,Z 991.277,A -85,B 0,C 180,E1 23997.086,E2 23997.086} C_VEL
LIN {X 0,Y 516.461,Z 965.817,A -85,B 0,C 180,E1 23996.435,E2 23996.435} C_VEL
LIN {X 0,Y 522.661,Z 883.056,A -85,B 0,C 180,E1 23994.631,E2 23994.631} C_VEL
LIN {X 0,Y 530.097,Z 807.65,A -85,B 0,C 180,E1 23992.871,E2 23992.871} C_VEL
LIN {X 0,Y 539.155,Z 734.139,A -85,B 0,C 180,E1 23991.079,E2 23991.079} C_VEL
LIN {X 0,Y 539.17,Z 719.766,A -85,B 0,C 180,E1 23990.299,E2 23990.299} C_VEL
LIN {X 0,Y 536.987,Z 712.812,A -85,B 0,C 180,E1 23989.314,E2 23989.314} C_VEL
LIN {X 0,Y 535.544,Z 708.614,A -85,B 0,C 180,E1 23988.56,E2 23988.56} C_VEL
LIN {X 0,Y 533.834,Z 703.537,A -85,B 0,C 180,E1 23987.403,E2 23987.403} C_VEL
LIN {X 0,Y 532.497,Z 699.7,A -85,B 0,C 180,E1 23985.988,E2 23985.988} C_VEL
LIN {X 0,Y 532.248,Z 697.384,A -85,B 0,C 180,E1 23984.448,E2 23984.448} C_VEL
LIN {X 0,Y 533.351,Z 697.623,A -85,B 0,C 180,E1 23982.701,E2 23982.701} C_VEL
LIN {X 0,Y 534.813,Z 699.472,A -85,B 0,C 180,E1 23981.585,E2 23981.585} C_VEL
LIN {X 0,Y 537.564,Z 703.659,A -85,B 0,C 180,E1 23980.177,E2 23980.177} C_VEL
LIN {X 0,Y 540.491,Z 708.87,A -85,B 0,C 180,E1 23979.037,E2 23979.037} C_VEL
LIN {X 0,Y 541.491,Z 711.346,A -85,B 0,C 180,E1 23978.662,E2 23978.662} C_VEL
LIN {X 0,Y 531.117,Z 789.734,A -85,B 0,C 180,E1 23976.747,E2 23976.747} C_VEL
LIN {X 0,Y 523.563,Z 862.181,A -85,B 0,C 180,E1 23975.045,E2 23975.045} C_VEL
LIN {X 0,Y 516.819,Z 947.194,A -85,B 0,C 180,E1 23973.126,E2 23973.126} C_VEL
LIN {X 0,Y 514.893,Z 969.84,A -85,B 0,C 180,E1 23972.412,E2 23972.412} C_VEL
LIN {X 0,Y 512.653,Z 991.899,A -85,B 0,C 180,E1 23971.516,E2 23971.516} C_VEL
LIN {X 0,Y 510.189,Z 1013.142,A -85,B 0,C 180,E1 23970.441,E2 23970.441} C_VEL
LIN {X 0,Y 507.675,Z 1032.797,A -85,B 0,C 180,E1 23969.241,E2 23969.241} C_VEL
LIN {X 0,Y 504.984,Z 1052.417,A -85,B 0,C 180,E1 23967.815,E2 23967.815} C_VEL
LIN {X 0,Y 502.396,Z 1070.271,A -85,B 0,C 180,E1 23966.287,E2 23966.287} C_VEL
LIN {X 0,Y 499.742,Z 1087.586,A -85,B 0,C 180,E1 23964.532,E2 23964.532} C_VEL
LIN {X 0,Y 497.259,Z 1103.483,A -85,B 0,C 180,E1 23962.636,E2 23962.636} C_VEL
LIN {X 0,Y 494.983,Z 1118.138,A -85,B 0,C 180,E1 23960.581,E2 23960.581} C_VEL
LIN {X 0,Y 493.161,Z 1130.422,A -85,B 0,C 180,E1 23958.564,E2 23958.564} C_VEL
LIN {X 0,Y 491.522,Z 1141.91,A -85,B 0,C 180,E1 23956.306,E2 23956.306} C_VEL
LIN {X 0,Y 490.276,Z 1151.482,A -85,B 0,C 180,E1 23954.048,E2 23954.048} C_VEL
LIN {X 0,Y 489.351,Z 1159.752,A -85,B 0,C 180,E1 23951.673,E2 23951.673} C_VEL
LIN {X 0,Y 488.732,Z 1166.23,A -85,B 0,C 180,E1 23949.304,E2 23949.304} C_VEL
LIN {X 0,Y 488.365,Z 1171.06,A -85,B 0,C 180,E1 23946.941,E2 23946.941} C_VEL
LIN {X 0,Y 488.171,Z 1174.553,A -85,B 0,C 180,E1 23944.466,E2 23944.466} C_VEL
LIN {X 0,Y 488.082,Z 1176.296,A -85,B 0,C 180,E1 23942.116,E2 23942.116} C_VEL
LIN {X 0,Y 488.057,Z 1176.576,A -85,B 0,C 180,E1 23939.65,E2 23939.65} C_VEL
LIN {X 0,Y 488.07,Z 1175.311,A -85,B 0,C 180,E1 23937.184,E2 23937.184} C_VEL
LIN {X 0,Y 488.138,Z 1172.308,A -85,B 0,C 180,E1 23934.714,E2 23934.714} C_VEL
LIN {X 0,Y 488.32,Z 1167.669,A -85,B 0,C 180,E1 23932.236,E2 23932.236} C_VEL
LIN {X 0,Y 488.692,Z 1161.431,A -85,B 0,C 180,E1 23929.789,E2 23929.789} C_VEL
LIN {X 0,Y 489.304,Z 1153.421,A -85,B 0,C 180,E1 23927.373,E2 23927.373} C_VEL
LIN {X 0,Y 490.168,Z 1144.151,A -85,B 0,C 180,E1 23925.109,E2 23925.109} C_VEL
LIN {X 0,Y 491.38,Z 1133.031,A -85,B 0,C 180,E1 23922.842,E2 23922.842} C_VEL
LIN {X 0,Y 492.889,Z 1120.489,A -85,B 0,C 180,E1 23920.694,E2 23920.694} C_VEL
LIN {X 0,Y 494.65,Z 1106.453,A -85,B 0,C 180,E1 23918.666,E2 23918.666} C_VEL
LIN {X 0,Y 496.696,Z 1090.792,A -85,B 0,C 180,E1 23916.732,E2 23916.732} C_VEL
LIN {X 0,Y 498.896,Z 1073.863,A -85,B 0,C 180,E1 23914.946,E2 23914.946} C_VEL
LIN {X 0,Y 501.189,Z 1055.827,A -85,B 0,C 180,E1 23913.331,E2 23913.331} C_VEL
LIN {X 0,Y 503.397,Z 1037.171,A -85,B 0,C 180,E1 23911.921,E2 23911.921} C_VEL
LIN {X 0,Y 505.63,Z 1017.005,A -85,B 0,C 180,E1 23910.635,E2 23910.635} C_VEL
LIN {X 0,Y 507.709,Z 996.067,A -85,B 0,C 180,E1 23909.531,E2 23909.531} C_VEL
LIN {X 0,Y 509.594,Z 973.958,A -85,B 0,C 180,E1 23908.599,E2 23908.599} C_VEL
LIN {X 0,Y 511.109,Z 951.946,A -85,B 0,C 180,E1 23907.887,E2 23907.887} C_VEL
LIN {X 0,Y 512.316,Z 928.666,A -85,B 0,C 180,E1 23907.34,E2 23907.34} C_VEL
LIN {X 0,Y 521.45,Z 696.363,A -85,B 0,C 180,E1 23903.378,E2 23903.378} C_VEL
LIN {X 0,Y 507.536,Z 671.029,A -85,B 0,C 180,E1 23901.843,E2 23901.843} C_VEL
LIN {X 0,Y 491.608,Z 643.565,A -85,B 0,C 180,E1 23900,E2 23900} C_VEL
LIN {X 0,Y 490.063,Z 640.193,A -85,B 0,C 180,E1 23899.796,E2 23899.796} C_VEL
LIN {X 0,Y 489.973,Z 639.632,A -85,B 0,C 180,E1 23899.75,E2 23899.75} C_VEL
LIN {X 0,Y 489.992,Z 639.629,A -85,B 0,C 180,E1 23896.234,E2 23896.234} C_VEL
LIN {X 0,Y 489.947,Z 639.637,A -85,B 0,C 180,E1 23892.724,E2 23892.724} C_VEL
LIN {X 0,Y 489.913,Z 639.642,A -85,B 0,C 180,E1 23889.15,E2 23889.15} C_VEL
LIN {X 0,Y 489.962,Z 639.632,A -85,B 0,C 180,E1 23885.693,E2 23885.693} C_VEL
LIN {X 0,Y 489.994,Z 639.63,A -85,B 0,C 180,E1 23882.183,E2 23882.183} C_VEL
LIN {X 0,Y 489.979,Z 639.636,A -85,B 0,C 180,E1 23878.658,E2 23878.658} C_VEL
LIN {X 0,Y 489.969,Z 639.637,A -85,B 0,C 180,E1 23875.118,E2 23875.118} C_VEL
LIN {X 0,Y 489.971,Z 639.633,A -85,B 0,C 180,E1 23871.552,E2 23871.552} C_VEL
LIN {X 0,Y 489.971,Z 639.629,A -85,B 0,C 180,E1 23867.949,E2 23867.949} C_VEL
LIN {X 0,Y 489.975,Z 639.631,A -85,B 0,C 180,E1 23864.418,E2 23864.418} C_VEL
LIN {X 0,Y 489.989,Z 639.634,A -85,B 0,C 180,E1 23860.822,E2 23860.822} C_VEL
LIN {X 0,Y 489.985,Z 639.628,A -85,B 0,C 180,E1 23859.344,E2 23859.344} C_VEL
LIN {X 0,Y 489.008,Z 639.751,A -85,B 0,C 180,E1 23858.444,E2 23858.444} C_VEL
LIN {X 0,Y 482.525,Z 640.562,A -85,B 0,C 180,E1 23855.912,E2 23855.912} C_VEL
LIN {X 0,Y 482.028,Z 640.626,A -85,B 0,C 180,E1 23855.251,E2 23855.251} C_VEL
LIN {X 0,Y 481.994,Z 640.616,A -85,B 0,C 180,E1 23851.666,E2 23851.666} C_VEL
LIN {X 0,Y 482.014,Z 640.623,A -85,B 0,C 180,E1 23848.219,E2 23848.219} C_VEL
LIN {X 0,Y 482.046,Z 640.612,A -85,B 0,C 180,E1 23844.61,E2 23844.61} C_VEL
LIN {X 0,Y 482.028,Z 640.619,A -85,B 0,C 180,E1 23841.172,E2 23841.172} C_VEL
LIN {X 0,Y 481.989,Z 640.617,A -85,B 0,C 180,E1 23837.664,E2 23837.664} C_VEL
LIN {X 0,Y 481.996,Z 640.625,A -85,B 0,C 180,E1 23834.11,E2 23834.11} C_VEL
LIN {X 0,Y 482.056,Z 640.619,A -85,B 0,C 180,E1 23830.619,E2 23830.619} C_VEL
LIN {X 0,Y 482.053,Z 640.62,A -85,B 0,C 180,E1 23827.05,E2 23827.05} C_VEL
LIN {X 0,Y 482.039,Z 640.626,A -85,B 0,C 180,E1 23823.374,E2 23823.374} C_VEL
LIN {X 0,Y 482.037,Z 640.625,A -85,B 0,C 180,E1 23819.871,E2 23819.871} C_VEL
LIN {X 0,Y 482.027,Z 640.627,A -85,B 0,C 180,E1 23816.228,E2 23816.228} C_VEL
LIN {X 0,Y 482.029,Z 640.626,A -85,B 0,C 180,E1 23812.723,E2 23812.723} C_VEL
LIN {X 0,Y 482.044,Z 640.622,A -85,B 0,C 180,E1 23809.205,E2 23809.205} C_VEL
LIN {X 0,Y 482.055,Z 640.732,A -85,B 0,C 180,E1 23806.02,E2 23806.02} C_VEL
LIN {X 0,Y 489.766,Z 666.749,A -85,B 0,C 180,E1 23803.307,E2 23803.307} C_VEL
LIN {X 0,Y 493.842,Z 682.103,A -85,B 0,C 180,E1 23801.765,E2 23801.765} C_VEL
LIN {X 0,Y 492.256,Z 725.624,A -85,B 0,C 180,E1 23798.129,E2 23798.129} C_VEL
LIN {X 0,Y 490.649,Z 767.274,A -85,B 0,C 180,E1 23794.647,E2 23794.647} C_VEL
LIN {X 0,Y 489.138,Z 809.394,A -85,B 0,C 180,E1 23791.14,E2 23791.14} C_VEL
LIN {X 0,Y 488.205,Z 837.982,A -85,B 0,C 180,E1 23788.799,E2 23788.799} C_VEL
LIN {X 0,Y 485.886,Z 981.98,A -85,B 0,C 180,E1 23786.229,E2 23786.229} C_VEL
LIN {X 0,Y 485.657,Z 998.693,A -85,B 0,C 180,E1 23785.712,E2 23785.712} C_VEL
LIN {X 0,Y 485.229,Z 1014.996,A -85,B 0,C 180,E1 23784.985,E2 23784.985} C_VEL
LIN {X 0,Y 484.695,Z 1030.619,A -85,B 0,C 180,E1 23784.04,E2 23784.04} C_VEL
LIN {X 0,Y 484.103,Z 1044.405,A -85,B 0,C 180,E1 23782.974,E2 23782.974} C_VEL
LIN {X 0,Y 483.452,Z 1057.75,A -85,B 0,C 180,E1 23781.68,E2 23781.68} C_VEL
LIN {X 0,Y 482.843,Z 1069.352,A -85,B 0,C 180,E1 23780.274,E2 23780.274} C_VEL
LIN {X 0,Y 482.28,Z 1080.033,A -85,B 0,C 180,E1 23778.66,E2 23778.66} C_VEL
LIN {X 0,Y 481.851,Z 1088.849,A -85,B 0,C 180,E1 23776.947,E2 23776.947} C_VEL
LIN {X 0,Y 481.582,Z 1095.478,A -85,B 0,C 180,E1 23775.286,E2 23775.286} C_VEL
LIN {X 0,Y 481.407,Z 1100.461,A -85,B 0,C 180,E1 23773.571,E2 23773.571} C_VEL
LIN {X 0,Y 481.36,Z 1104.074,A -85,B 0,C 180,E1 23771.743,E2 23771.743} C_VEL
LIN {X 0,Y 481.431,Z 1105.917,A -85,B 0,C 180,E1 23769.924,E2 23769.924} C_VEL
LIN {X 0,Y 481.623,Z 1106.002,A -85,B 0,C 180,E1 23767.993,E2 23767.993} C_VEL
LIN {X 0,Y 481.947,Z 1104.369,A -85,B 0,C 180,E1 23766.191,E2 23766.191} C_VEL
LIN {X 0,Y 482.445,Z 1100.694,A -85,B 0,C 180,E1 23764.276,E2 23764.276} C_VEL
LIN {X 0,Y 483.079,Z 1095.382,A -85,B 0,C 180,E1 23762.489,E2 23762.489} C_VEL
LIN {X 0,Y 483.907,Z 1088.036,A -85,B 0,C 180,E1 23760.708,E2 23760.708} C_VEL
LIN {X 0,Y 484.802,Z 1079.759,A -85,B 0,C 180,E1 23759.17,E2 23759.17} C_VEL
LIN {X 0,Y 485.838,Z 1069.271,A -85,B 0,C 180,E1 23757.638,E2 23757.638} C_VEL
LIN {X 0,Y 486.816,Z 1058.201,A -85,B 0,C 180,E1 23756.347,E2 23756.347} C_VEL
LIN {X 0,Y 487.85,Z 1044.306,A -85,B 0,C 180,E1 23755.059,E2 23755.059} C_VEL
LIN {X 0,Y 488.694,Z 1029.739,A -85,B 0,C 180,E1 23754.008,E2 23754.008} C_VEL
LIN {X 0,Y 489.296,Z 1016.503,A -85,B 0,C 180,E1 23753.27,E2 23753.27} C_VEL
LIN {X 0,Y 489.723,Z 1004.074,A -85,B 0,C 180,E1 23752.725,E2 23752.725} C_VEL
LIN {X 0,Y 490.026,Z 989.447,A -85,B 0,C 180,E1 23752.243,E2 23752.243} C_VEL
LIN {X 0,Y 490.647,Z 950.171,A -85,B 0,C 180,E1 23751.457,E2 23751.457} C_VEL
LIN {X 0,Y 494.22,Z 848.117,A -85,B 0,C 180,E1 23749.447,E2 23749.447} C_VEL
LIN {X 0,Y 494.732,Z 844.409,A -85,B 0,C 180,E1 23749.164,E2 23749.164} C_VEL
LIN {X 0,Y 496.941,Z 797.868,A -85,B 0,C 180,E1 23745.312,E2 23745.312} C_VEL
LIN {X 0,Y 498.972,Z 754.096,A -85,B 0,C 180,E1 23741.721,E2 23741.721} C_VEL
LIN {X 0,Y 500.954,Z 713.166,A -85,B 0,C 180,E1 23738.39,E2 23738.39} C_VEL
LIN {X 0,Y 502.146,Z 689.458,A -85,B 0,C 180,E1 23736.467,E2 23736.467} C_VEL
LIN {X 0,Y 498.439,Z 676.832,A -85,B 0,C 180,E1 23734.956,E2 23734.956} C_VEL
LIN {X 0,Y 492.701,Z 661.998,A -85,B 0,C 180,E1 23732.918,E2 23732.918} C_VEL
LIN {X 0,Y 486.997,Z 650.162,A -85,B 0,C 180,E1 23730.999,E2 23730.999} C_VEL
LIN {X 0,Y 485.002,Z 646.616,A -85,B 0,C 180,E1 23730.342,E2 23730.342} C_VEL
LIN {X 0,Y 484.359,Z 645.31,A -85,B 0,C 180,E1 23730.11,E2 23730.11} C_VEL
LIN {X 0,Y 482.409,Z 642.167,A -85,B 0,C 180,E1 23729.48,E2 23729.48} C_VEL
LIN {X 0,Y 482.055,Z 640.621,A -85,B 0,C 180,E1 23729.248,E2 23729.248} C_VEL
LIN {X 0,Y 482.057,Z 640.622,A -85,B 0,C 180,E1 23725.508,E2 23725.508} C_VEL
LIN {X 0,Y 482.054,Z 640.62,A -85,B 0,C 180,E1 23721.819,E2 23721.819} C_VEL
LIN {X 0,Y 482.026,Z 640.625,A -85,B 0,C 180,E1 23718.129,E2 23718.129} C_VEL
LIN {X 0,Y 482.069,Z 640.772,A -85,B 0,C 180,E1 23715.318,E2 23715.318} C_VEL
LIN {X 0,Y 489.573,Z 663.008,A -85,B 0,C 180,E1 23711.899,E2 23711.899} C_VEL
LIN {X 0,Y 493.868,Z 676.112,A -85,B 0,C 180,E1 23710.041,E2 23710.041} C_VEL
LIN {X 0,Y 510.343,Z 709.201,A -85,B 0,C 180,E1 23708.057,E2 23708.057} C_VEL
LIN {X 0,Y 514.53,Z 733.357,A -85,B 0,C 180,E1 23707.254,E2 23707.254} C_VEL
LIN {X 0,Y 505.028,Z 965.238,A -85,B 0,C 180,E1 23703.216,E2 23703.216} C_VEL
LIN {X 0,Y 503.796,Z 989.367,A -85,B 0,C 180,E1 23702.721,E2 23702.721} C_VEL
LIN {X 0,Y 502.039,Z 1012.829,A -85,B 0,C 180,E1 23702.034,E2 23702.034} C_VEL
LIN {X 0,Y 500.064,Z 1034.665,A -85,B 0,C 180,E1 23701.187,E2 23701.187} C_VEL
LIN {X 0,Y 497.84,Z 1056.178,A -85,B 0,C 180,E1 23700.138,E2 23700.138} C_VEL
LIN {X 0,Y 495.473,Z 1076.67,A -85,B 0,C 180,E1 23698.9,E2 23698.9} C_VEL
LIN {X 0,Y 493.026,Z 1096.406,A -85,B 0,C 180,E1 23697.474,E2 23697.474} C_VEL
LIN {X 0,Y 490.6,Z 1115.303,A -85,B 0,C 180,E1 23695.856,E2 23695.856} C_VEL
LIN {X 0,Y 488.334,Z 1132.696,A -85,B 0,C 180,E1 23694.108,E2 23694.108} C_VEL
LIN {X 0,Y 486.213,Z 1148.958,A -85,B 0,C 180,E1 23692.177,E2 23692.177} C_VEL
LIN {X 0,Y 484.421,Z 1163.42,A -85,B 0,C 180,E1 23690.162,E2 23690.162} C_VEL
LIN {X 0,Y 482.883,Z 1176.853,A -85,B 0,C 180,E1 23687.969,E2 23687.969} C_VEL
LIN {X 0,Y 481.743,Z 1188.249,A -85,B 0,C 180,E1 23685.775,E2 23685.775} C_VEL
LIN {X 0,Y 480.914,Z 1198.182,A -85,B 0,C 180,E1 23683.464,E2 23683.464} C_VEL
LIN {X 0,Y 480.382,Z 1206.743,A -85,B 0,C 180,E1 23681.038,E2 23681.038} C_VEL
LIN {X 0,Y 480.123,Z 1213.519,A -85,B 0,C 180,E1 23678.622,E2 23678.622} C_VEL
LIN {X 0,Y 480.034,Z 1218.448,A -85,B 0,C 180,E1 23676.216,E2 23676.216} C_VEL
LIN {X 0,Y 480.042,Z 1221.933,A -85,B 0,C 180,E1 23673.701,E2 23673.701} C_VEL
LIN {X 0,Y 480.057,Z 1223.601,A -85,B 0,C 180,E1 23671.431,E2 23671.431} C_VEL
LIN {X 0,Y 480.067,Z 1223.772,A -85,B 0,C 180,E1 23669.044,E2 23669.044} C_VEL
LIN {X 0,Y 480.03,Z 1222.472,A -85,B 0,C 180,E1 23666.655,E2 23666.655} C_VEL
LIN {X 0,Y 480.013,Z 1219.475,A -85,B 0,C 180,E1 23664.26,E2 23664.26} C_VEL
LIN {X 0,Y 480.09,Z 1214.68,A -85,B 0,C 180,E1 23661.736,E2 23661.736} C_VEL
LIN {X 0,Y 480.321,Z 1208.418,A -85,B 0,C 180,E1 23659.322,E2 23659.322} C_VEL
LIN {X 0,Y 480.82,Z 1200.291,A -85,B 0,C 180,E1 23656.897,E2 23656.897} C_VEL
LIN {X 0,Y 481.721,Z 1189.719,A -85,B 0,C 180,E1 23654.344,E2 23654.344} C_VEL
LIN {X 0,Y 482.951,Z 1178.161,A -85,B 0,C 180,E1 23652.031,E2 23652.031} C_VEL
LIN {X 0,Y 484.535,Z 1165.127,A -85,B 0,C 180,E1 23649.84,E2 23649.84} C_VEL
LIN {X 0,Y 486.435,Z 1150.702,A -85,B 0,C 180,E1 23647.775,E2 23647.775} C_VEL
LIN {X 0,Y 488.813,Z 1133.928,A -85,B 0,C 180,E1 23645.721,E2 23645.721} C_VEL
LIN {X 0,Y 491.41,Z 1116.131,A -85,B 0,C 180,E1 23643.862,E2 23643.862} C_VEL
LIN {X 0,Y 494.24,Z 1096.667,A -85,B 0,C 180,E1 23642.137,E2 23642.137} C_VEL
LIN {X 0,Y 497.04,Z 1077.065,A -85,B 0,C 180,E1 23640.668,E2 23640.668} C_VEL
LIN {X 0,Y 500.021,Z 1055.52,A -85,B 0,C 180,E1 23639.305,E2 23639.305} C_VEL
LIN {X 0,Y 502.985,Z 1033.339,A -85,B 0,C 180,E1 23638.142,E2 23638.142} C_VEL
LIN {X 0,Y 505.825,Z 1010.463,A -85,B 0,C 180,E1 23637.167,E2 23637.167} C_VEL
LIN {X 0,Y 508.664,Z 985.366,A -85,B 0,C 180,E1 23636.338,E2 23636.338} C_VEL
LIN {X 0,Y 511.125,Z 957.392,A -85,B 0,C 180,E1 23635.65,E2 23635.65} C_VEL
LIN {X 0,Y 517.279,Z 883.532,A -85,B 0,C 180,E1 23633.98,E2 23633.98} C_VEL
LIN {X 0,Y 525.426,Z 808.485,A -85,B 0,C 180,E1 23632.172,E2 23632.172} C_VEL
LIN {X 0,Y 535.176,Z 736.115,A -85,B 0,C 180,E1 23630.361,E2 23630.361} C_VEL
LIN {X 0,Y 535.448,Z 724.611,A -85,B 0,C 180,E1 23629.716,E2 23629.716} C_VEL
LIN {X 0,Y 533.366,Z 717.062,A -85,B 0,C 180,E1 23628.565,E2 23628.565} C_VEL
LIN {X 0,Y 531.41,Z 710.729,A -85,B 0,C 180,E1 23627.13,E2 23627.13} C_VEL
LIN {X 0,Y 530.349,Z 707.161,A -85,B 0,C 180,E1 23625.763,E2 23625.763} C_VEL
LIN {X 0,Y 530.27,Z 705.122,A -85,B 0,C 180,E1 23624.384,E2 23624.384} C_VEL
LIN {X 0,Y 531.436,Z 705.407,A -85,B 0,C 180,E1 23622.636,E2 23622.636} C_VEL
LIN {X 0,Y 533.093,Z 707.852,A -85,B 0,C 180,E1 23621.386,E2 23621.386} C_VEL
LIN {X 0,Y 535.119,Z 711.265,A -85,B 0,C 180,E1 23620.326,E2 23620.326} C_VEL
LIN {X 0,Y 537.482,Z 715.752,A -85,B 0,C 180,E1 23619.336,E2 23619.336} C_VEL
LIN {X 0,Y 526.355,Z 793.108,A -85,B 0,C 180,E1 23617.4,E2 23617.4} C_VEL
LIN {X 0,Y 518.276,Z 863.569,A -85,B 0,C 180,E1 23615.691,E2 23615.691} C_VEL
LIN {X 0,Y 510.85,Z 948.217,A -85,B 0,C 180,E1 23613.709,E2 23613.709} C_VEL
LIN {X 0,Y 508.695,Z 971.27,A -85,B 0,C 180,E1 23612.957,E2 23612.957} C_VEL
LIN {X 0,Y 506.255,Z 993.5,A -85,B 0,C 180,E1 23612.028,E2 23612.028} C_VEL
LIN {X 0,Y 503.401,Z 1016.382,A -85,B 0,C 180,E1 23610.83,E2 23610.83} C_VEL
LIN {X 0,Y 500.64,Z 1036.254,A -85,B 0,C 180,E1 23609.561,E2 23609.561} C_VEL
LIN {X 0,Y 497.782,Z 1055.474,A -85,B 0,C 180,E1 23608.104,E2 23608.104} C_VEL
LIN {X 0,Y 494.81,Z 1074.466,A -85,B 0,C 180,E1 23606.398,E2 23606.398} C_VEL
LIN {X 0,Y 492.078,Z 1091.275,A -85,B 0,C 180,E1 23604.619,E2 23604.619} C_VEL
LIN {X 0,Y 489.405,Z 1107.534,A -85,B 0,C 180,E1 23602.59,E2 23602.59} C_VEL
LIN {X 0,Y 487.002,Z 1122.054,A -85,B 0,C 180,E1 23600.431,E2 23600.431} C_VEL
LIN {X 0,Y 485.035,Z 1134.35,A -85,B 0,C 180,E1 23598.263,E2 23598.263} C_VEL
LIN {X 0,Y 483.403,Z 1145.311,A -85,B 0,C 180,E1 23595.97,E2 23595.97} C_VEL
LIN {X 0,Y 482.143,Z 1154.867,A -85,B 0,C 180,E1 23593.555,E2 23593.555} C_VEL
LIN {X 0,Y 481.243,Z 1162.456,A -85,B 0,C 180,E1 23591.144,E2 23591.144} C_VEL
LIN {X 0,Y 480.65,Z 1168.646,A -85,B 0,C 180,E1 23588.617,E2 23588.617} C_VEL
LIN {X 0,Y 480.326,Z 1172.979,A -85,B 0,C 180,E1 23586.217,E2 23586.217} C_VEL
LIN {X 0,Y 480.156,Z 1175.684,A -85,B 0,C 180,E1 23583.823,E2 23583.823} C_VEL
LIN {X 0,Y 480.091,Z 1177.019,A -85,B 0,C 180,E1 23581.196,E2 23581.196} C_VEL
LIN {X 0,Y 480.068,Z 1176.726,A -85,B 0,C 180,E1 23578.743,E2 23578.743} C_VEL
LIN {X 0,Y 480.091,Z 1174.773,A -85,B 0,C 180,E1 23576.301,E2 23576.301} C_VEL
LIN {X 0,Y 480.191,Z 1171.209,A -85,B 0,C 180,E1 23573.787,E2 23573.787} C_VEL
LIN {X 0,Y 480.445,Z 1166.13,A -85,B 0,C 180,E1 23571.328,E2 23571.328} C_VEL
LIN {X 0,Y 480.9,Z 1159.188,A -85,B 0,C 180,E1 23568.854,E2 23568.854} C_VEL
LIN {X 0,Y 481.636,Z 1150.655,A -85,B 0,C 180,E1 23566.435,E2 23566.435} C_VEL
LIN {X 0,Y 482.665,Z 1140.774,A -85,B 0,C 180,E1 23564.133,E2 23564.133} C_VEL
LIN {X 0,Y 484.052,Z 1128.917,A -85,B 0,C 180,E1 23561.845,E2 23561.845} C_VEL
LIN {X 0,Y 485.66,Z 1116.152,A -85,B 0,C 180,E1 23559.767,E2 23559.767} C_VEL
LIN {X 0,Y 487.631,Z 1101.361,A -85,B 0,C 180,E1 23557.71,E2 23557.71} C_VEL
LIN {X 0,Y 489.705,Z 1086.002,A -85,B 0,C 180,E1 23555.882,E2 23555.882} C_VEL
LIN {X 0,Y 491.971,Z 1068.927,A -85,B 0,C 180,E1 23554.157,E2 23554.157} C_VEL
LIN {X 0,Y 494.366,Z 1050.163,A -85,B 0,C 180,E1 23552.542,E2 23552.542} C_VEL
LIN {X 0,Y 496.735,Z 1030.525,A -85,B 0,C 180,E1 23551.115,E2 23551.115} C_VEL
LIN {X 0,Y 499.001,Z 1010.089,A -85,B 0,C 180,E1 23549.875,E2 23549.875} C_VEL
LIN {X 0,Y 501.076,Z 988.566,A -85,B 0,C 180,E1 23548.817,E2 23548.817} C_VEL
LIN {X 0,Y 502.869,Z 966.561,A -85,B 0,C 180,E1 23547.956,E2 23547.956} C_VEL
LIN {X 0,Y 504.369,Z 943.377,A -85,B 0,C 180,E1 23547.268,E2 23547.268} C_VEL
LIN {X 0,Y 505.51,Z 919.884,A -85,B 0,C 180,E1 23546.781,E2 23546.781} C_VEL
LIN {X 0,Y 514.22,Z 706.961,A -85,B 0,C 180,E1 23543.091,E2 23543.091} C_VEL
LIN {X 0,Y 514.446,Z 698.774,A -85,B 0,C 180,E1 23542.936,E2 23542.936} C_VEL
LIN {X 0,Y 496.928,Z 667.287,A -85,B 0,C 180,E1 23540.96,E2 23540.96} C_VEL
LIN {X 0,Y 483.624,Z 644.484,A -85,B 0,C 180,E1 23539.357,E2 23539.357} C_VEL
LIN {X 0,Y 482.127,Z 641.089,A -85,B 0,C 180,E1 23539.152,E2 23539.152} C_VEL
LIN {X 0,Y 482.055,Z 640.623,A -85,B 0,C 180,E1 23539.133,E2 23539.133} C_VEL
LIN {X 0,Y 482.043,Z 640.626,A -85,B 0,C 180,E1 23535.489,E2 23535.489} C_VEL
LIN {X 0,Y 482.04,Z 640.623,A -85,B 0,C 180,E1 23531.875,E2 23531.875} C_VEL
LIN {X 0,Y 482.016,Z 640.626,A -85,B 0,C 180,E1 23528.335,E2 23528.335} C_VEL
LIN {X 0,Y 482.023,Z 640.621,A -85,B 0,C 180,E1 23524.776,E2 23524.776} C_VEL
LIN {X 0,Y 482.039,Z 640.623,A -85,B 0,C 180,E1 23521.238,E2 23521.238} C_VEL
LIN {X 0,Y 482.064,Z 640.622,A -85,B 0,C 180,E1 23517.673,E2 23517.673} C_VEL
LIN {X 0,Y 482.009,Z 640.629,A -85,B 0,C 180,E1 23514.122,E2 23514.122} C_VEL
LIN {X 0,Y 481.976,Z 640.631,A -85,B 0,C 180,E1 23510.525,E2 23510.525} C_VEL
LIN {X 0,Y 482.015,Z 640.622,A -85,B 0,C 180,E1 23506.884,E2 23506.884} C_VEL
LIN {X 0,Y 482.052,Z 640.61,A -85,B 0,C 180,E1 23503.313,E2 23503.313} C_VEL
LIN {X 0,Y 482.032,Z 640.618,A -85,B 0,C 180,E1 23499.674,E2 23499.674} C_VEL
LIN {X 0,Y 481.994,Z 640.628,A -85,B 0,C 180,E1 23496.075,E2 23496.075} C_VEL
LIN {X 0,Y 482.028,Z 640.626,A -85,B 0,C 180,E1 23495.251,E2 23495.251} C_VEL
LIN {X 0,Y 481.082,Z 640.747,A -85,B 0,C 180,E1 23494.336,E2 23494.336} C_VEL
LIN {X 0,Y 474.522,Z 641.548,A -85,B 0,C 180,E1 23491.695,E2 23491.695} C_VEL
LIN {X 0,Y 474.104,Z 641.607,A -85,B 0,C 180,E1 23491.09,E2 23491.09} C_VEL
LIN {X 0,Y 474.104,Z 641.604,A -85,B 0,C 180,E1 23487.584,E2 23487.584} C_VEL
LIN {X 0,Y 474.112,Z 641.606,A -85,B 0,C 180,E1 23483.949,E2 23483.949} C_VEL
LIN {X 0,Y 474.108,Z 641.602,A -85,B 0,C 180,E1 23480.288,E2 23480.288} C_VEL
LIN {X 0,Y 474.096,Z 641.606,A -85,B 0,C 180,E1 23476.587,E2 23476.587} C_VEL
LIN {X 0,Y 474.082,Z 641.613,A -85,B 0,C 180,E1 23472.954,E2 23472.954} C_VEL
LIN {X 0,Y 474.095,Z 641.611,A -85,B 0,C 180,E1 23469.379,E2 23469.379} C_VEL
LIN {X 0,Y 474.111,Z 641.608,A -85,B 0,C 180,E1 23465.851,E2 23465.851} C_VEL
LIN {X 0,Y 474.112,Z 641.61,A -85,B 0,C 180,E1 23462.222,E2 23462.222} C_VEL
LIN {X 0,Y 474.049,Z 641.618,A -85,B 0,C 180,E1 23458.746,E2 23458.746} C_VEL
LIN {X 0,Y 474.051,Z 641.617,A -85,B 0,C 180,E1 23455.128,E2 23455.128} C_VEL
LIN {X 0,Y 474.089,Z 641.612,A -85,B 0,C 180,E1 23451.481,E2 23451.481} C_VEL
LIN {X 0,Y 474.114,Z 641.609,A -85,B 0,C 180,E1 23447.886,E2 23447.886} C_VEL
LIN {X 0,Y 474.108,Z 641.723,A -85,B 0,C 180,E1 23446.402,E2 23446.402} C_VEL
LIN {X 0,Y 481.74,Z 667.236,A -85,B 0,C 180,E1 23443.718,E2 23443.718} C_VEL
LIN {X 0,Y 486.309,Z 684.221,A -85,B 0,C 180,E1 23441.984,E2 23441.984} C_VEL
LIN {X 0,Y 484.624,Z 727.614,A -85,B 0,C 180,E1 23438.32,E2 23438.32} C_VEL
LIN {X 0,Y 482.995,Z 769.077,A -85,B 0,C 180,E1 23434.842,E2 23434.842} C_VEL
LIN {X 0,Y 481.445,Z 810.77,A -85,B 0,C 180,E1 23431.345,E2 23431.345} C_VEL
LIN {X 0,Y 480.485,Z 838.781,A -85,B 0,C 180,E1 23429.03,E2 23429.03} C_VEL
LIN {X 0,Y 478.046,Z 982.564,A -85,B 0,C 180,E1 23426.409,E2 23426.409} C_VEL
LIN {X 0,Y 477.816,Z 998.951,A -85,B 0,C 180,E1 23425.898,E2 23425.898} C_VEL
LIN {X 0,Y 477.376,Z 1015.412,A -85,B 0,C 180,E1 23425.16,E2 23425.16} C_VEL
LIN {X 0,Y 476.821,Z 1031.162,A -85,B 0,C 180,E1 23424.196,E2 23424.196} C_VEL
LIN {X 0,Y 476.214,Z 1045.013,A -85,B 0,C 180,E1 23423.115,E2 23423.115} C_VEL
LIN {X 0,Y 475.533,Z 1058.584,A -85,B 0,C 180,E1 23421.781,E2 23421.781} C_VEL
LIN {X 0,Y 474.95,Z 1069.498,A -85,B 0,C 180,E1 23420.452,E2 23420.452} C_VEL
LIN {X 0,Y 474.361,Z 1080.323,A -85,B 0,C 180,E1 23418.811,E2 23418.811} C_VEL
LIN {X 0,Y 473.937,Z 1088.833,A -85,B 0,C 180,E1 23417.176,E2 23417.176} C_VEL
LIN {X 0,Y 473.624,Z 1096.365,A -85,B 0,C 180,E1 23415.298,E2 23415.298} C_VEL
LIN {X 0,Y 473.449,Z 1101.392,A -85,B 0,C 180,E1 23413.555,E2 23413.555} C_VEL
LIN {X 0,Y 473.41,Z 1105.038,A -85,B 0,C 180,E1 23411.696,E2 23411.696} C_VEL
LIN {X 0,Y 473.493,Z 1106.906,A -85,B 0,C 180,E1 23409.846,E2 23409.846} C_VEL
LIN {X 0,Y 473.707,Z 1107.011,A -85,B 0,C 180,E1 23407.883,E2 23407.883} C_VEL
LIN {X 0,Y 474.061,Z 1105.384,A -85,B 0,C 180,E1 23406.051,E2 23406.051} C_VEL
LIN {X 0,Y 474.6,Z 1101.73,A -85,B 0,C 180,E1 23404.105,E2 23404.105} C_VEL
LIN {X 0,Y 475.291,Z 1096.445,A -85,B 0,C 180,E1 23402.288,E2 23402.288} C_VEL
LIN {X 0,Y 476.182,Z 1089.099,A -85,B 0,C 180,E1 23400.479,E2 23400.479} C_VEL
LIN {X 0,Y 477.136,Z 1080.806,A -85,B 0,C 180,E1 23398.917,E2 23398.917} C_VEL
LIN {X 0,Y 478.236,Z 1070.29,A -85,B 0,C 180,E1 23397.361,E2 23397.361} C_VEL
LIN {X 0,Y 479.322,Z 1058.637,A -85,B 0,C 180,E1 23395.99,E2 23395.99} C_VEL
LIN {X 0,Y 480.384,Z 1045.385,A -85,B 0,C 180,E1 23394.743,E2 23394.743} C_VEL
LIN {X 0,Y 481.238,Z 1031.781,A -85,B 0,C 180,E1 23393.735,E2 23393.735} C_VEL
LIN {X 0,Y 481.892,Z 1018.404,A -85,B 0,C 180,E1 23392.966,E2 23392.966} C_VEL
LIN {X 0,Y 482.365,Z 1005.585,A -85,B 0,C 180,E1 23392.389,E2 23392.389} C_VEL
LIN {X 0,Y 482.696,Z 990.753,A -85,B 0,C 180,E1 23391.889,E2 23391.889} C_VEL
LIN {X 0,Y 483.388,Z 951.016,A -85,B 0,C 180,E1 23391.069,E2 23391.069} C_VEL
LIN {X 0,Y 487.257,Z 849.004,A -85,B 0,C 180,E1 23388.996,E2 23388.996} C_VEL
LIN {X 0,Y 487.846,Z 842.521,A -85,B 0,C 180,E1 23388.47,E2 23388.47} C_VEL
LIN {X 0,Y 489.966,Z 800.659,A -85,B 0,C 180,E1 23384.977,E2 23384.977} C_VEL
LIN {X 0,Y 492.153,Z 758.395,A -85,B 0,C 180,E1 23381.458,E2 23381.458} C_VEL
LIN {X 0,Y 494.507,Z 715.385,A -85,B 0,C 180,E1 23377.906,E2 23377.906} C_VEL
LIN {X 0,Y 495.663,Z 692.659,A -85,B 0,C 180,E1 23376.033,E2 23376.033} C_VEL
LIN {X 0,Y 491.973,Z 680.092,A -85,B 0,C 180,E1 23374.468,E2 23374.468} C_VEL
LIN {X 0,Y 486.997,Z 667.069,A -85,B 0,C 180,E1 23372.616,E2 23372.616} C_VEL
LIN {X 0,Y 481.528,Z 655.663,A -85,B 0,C 180,E1 23370.702,E2 23370.702} C_VEL
LIN {X 0,Y 478.972,Z 650.908,A -85,B 0,C 180,E1 23369.792,E2 23369.792} C_VEL
LIN {X 0,Y 477.149,Z 647.099,A -85,B 0,C 180,E1 23369.059,E2 23369.059} C_VEL
LIN {X 0,Y 474.641,Z 643.693,A -85,B 0,C 180,E1 23368.218,E2 23368.218} C_VEL
LIN {X 0,Y 474.101,Z 641.612,A -85,B 0,C 180,E1 23367.828,E2 23367.828} C_VEL
LIN {X 0,Y 474.095,Z 641.615,A -85,B 0,C 180,E1 23364.251,E2 23364.251} C_VEL
LIN {X 0,Y 474.115,Z 641.609,A -85,B 0,C 180,E1 23360.519,E2 23360.519} C_VEL
LIN {X 0,Y 474.109,Z 641.605,A -85,B 0,C 180,E1 23356.682,E2 23356.682} C_VEL
LIN {X 0,Y 474.103,Z 641.625,A -85,B 0,C 180,E1 23355.938,E2 23355.938} C_VEL
LIN {X 0,Y 481.641,Z 663.986,A -85,B 0,C 180,E1 23352.428,E2 23352.428} C_VEL
LIN {X 0,Y 485.512,Z 675.724,A -85,B 0,C 180,E1 23350.72,E2 23350.72} C_VEL
LIN {X 0,Y 503.16,Z 710.966,A -85,B 0,C 180,E1 23348.556,E2 23348.556} C_VEL
LIN {X 0,Y 504.183,Z 713.876,A -85,B 0,C 180,E1 23348.416,E2 23348.416} C_VEL
LIN {X 0,Y 507.695,Z 734.76,A -85,B 0,C 180,E1 23347.709,E2 23347.709} C_VEL
LIN {X 0,Y 497.06,Z 981.73,A -85,B 0,C 180,E1 23343.295,E2 23343.295} C_VEL
LIN {X 0,Y 495.357,Z 1005.254,A -85,B 0,C 180,E1 23342.666,E2 23342.666} C_VEL
LIN {X 0,Y 493.413,Z 1027.286,A -85,B 0,C 180,E1 23341.861,E2 23341.861} C_VEL
LIN {X 0,Y 491.174,Z 1048.89,A -85,B 0,C 180,E1 23340.861,E2 23340.861} C_VEL
LIN {X 0,Y 488.784,Z 1069.779,A -85,B 0,C 180,E1 23339.671,E2 23339.671} C_VEL
LIN {X 0,Y 486.248,Z 1090.213,A -85,B 0,C 180,E1 23338.262,E2 23338.262} C_VEL
LIN {X 0,Y 483.668,Z 1109.624,A -85,B 0,C 180,E1 23336.652,E2 23336.652} C_VEL
LIN {X 0,Y 481.306,Z 1127.115,A -85,B 0,C 180,E1 23334.941,E2 23334.941} C_VEL
LIN {X 0,Y 478.999,Z 1144.259,A -85,B 0,C 180,E1 23332.974,E2 23332.974} C_VEL
LIN {X 0,Y 477.088,Z 1159.005,A -85,B 0,C 180,E1 23330.999,E2 23330.999} C_VEL
LIN {X 0,Y 475.416,Z 1172.668,A -85,B 0,C 180,E1 23328.834,E2 23328.834} C_VEL
LIN {X 0,Y 474.091,Z 1184.917,A -85,B 0,C 180,E1 23326.54,E2 23326.54} C_VEL
LIN {X 0,Y 473.13,Z 1195.463,A -85,B 0,C 180,E1 23324.189,E2 23324.189} C_VEL
LIN {X 0,Y 472.515,Z 1204.118,A -85,B 0,C 180,E1 23321.843,E2 23321.843} C_VEL
LIN {X 0,Y 472.175,Z 1211.32,A -85,B 0,C 180,E1 23319.383,E2 23319.383} C_VEL
LIN {X 0,Y 472.044,Z 1216.831,A -85,B 0,C 180,E1 23316.933,E2 23316.933} C_VEL
LIN {X 0,Y 472.036,Z 1220.476,A -85,B 0,C 180,E1 23314.615,E2 23314.615} C_VEL
LIN {X 0,Y 472.074,Z 1222.826,A -85,B 0,C 180,E1 23312.062,E2 23312.062} C_VEL
LIN {X 0,Y 472.071,Z 1223.517,A -85,B 0,C 180,E1 23309.634,E2 23309.634} C_VEL
LIN {X 0,Y 472.048,Z 1222.507,A -85,B 0,C 180,E1 23307.206,E2 23307.206} C_VEL
LIN {X 0,Y 472.017,Z 1219.839,A -85,B 0,C 180,E1 23304.649,E2 23304.649} C_VEL
LIN {X 0,Y 472.052,Z 1215.891,A -85,B 0,C 180,E1 23302.33,E2 23302.33} C_VEL
LIN {X 0,Y 472.258,Z 1209.777,A -85,B 0,C 180,E1 23299.754,E2 23299.754} C_VEL
LIN {X 0,Y 472.718,Z 1202.205,A -85,B 0,C 180,E1 23297.291,E2 23297.291} C_VEL
LIN {X 0,Y 473.475,Z 1193.201,A -85,B 0,C 180,E1 23294.943,E2 23294.943} C_VEL
LIN {X 0,Y 474.631,Z 1182.356,A -85,B 0,C 180,E1 23292.592,E2 23292.592} C_VEL
LIN {X 0,Y 476.144,Z 1170.233,A -85,B 0,C 180,E1 23290.365,E2 23290.365} C_VEL
LIN {X 0,Y 478.116,Z 1155.894,A -85,B 0,C 180,E1 23288.144,E2 23288.144} C_VEL
LIN {X 0,Y 480.367,Z 1140.54,A -85,B 0,C 180,E1 23286.117,E2 23286.117} C_VEL
LIN {X 0,Y 483.092,Z 1122.735,A -85,B 0,C 180,E1 23284.104,E2 23284.104} C_VEL
LIN {X 0,Y 485.937,Z 1104.659,A -85,B 0,C 180,E1 23282.359,E2 23282.359} C_VEL
LIN {X 0,Y 489.091,Z 1084.186,A -85,B 0,C 180,E1 23280.682,E2 23280.682} C_VEL
LIN {X 0,Y 492.308,Z 1062.737,A -85,B 0,C 180,E1 23279.214,E2 23279.214} C_VEL
LIN {X 0,Y 495.515,Z 1040.488,A -85,B 0,C 180,E1 23277.946,E2 23277.946} C_VEL
LIN {X 0,Y 498.725,Z 1016.929,A -85,B 0,C 180,E1 23276.851,E2 23276.851} C_VEL
LIN {X 0,Y 501.846,Z 992.079,A -85,B 0,C 180,E1 23275.943,E2 23275.943} C_VEL
LIN {X 0,Y 504.702,Z 965.08,A -85,B 0,C 180,E1 23275.2,E2 23275.2} C_VEL
LIN {X 0,Y 512.072,Z 884.756,A -85,B 0,C 180,E1 23273.316,E2 23273.316} C_VEL
LIN {X 0,Y 520.955,Z 810.098,A -85,B 0,C 180,E1 23271.463,E2 23271.463} C_VEL
LIN {X 0,Y 531.523,Z 738.312,A -85,B 0,C 180,E1 23269.628,E2 23269.628} C_VEL
LIN {X 0,Y 531.938,Z 729.556,A -85,B 0,C 180,E1 23269.121,E2 23269.121} C_VEL
LIN {X 0,Y 530.295,Z 722.94,A -85,B 0,C 180,E1 23268.022,E2 23268.022} C_VEL
LIN {X 0,Y 528.977,Z 717.677,A -85,B 0,C 180,E1 23266.778,E2 23266.778} C_VEL
LIN {X 0,Y 528.235,Z 714.623,A -85,B 0,C 180,E1 23265.532,E2 23265.532} C_VEL
LIN {X 0,Y 528.295,Z 712.858,A -85,B 0,C 180,E1 23264.301,E2 23264.301} C_VEL
LIN {X 0,Y 529.379,Z 713.129,A -85,B 0,C 180,E1 23262.696,E2 23262.696} C_VEL
LIN {X 0,Y 530.943,Z 715.678,A -85,B 0,C 180,E1 23261.449,E2 23261.449} C_VEL
LIN {X 0,Y 532.628,Z 718.733,A -85,B 0,C 180,E1 23260.508,E2 23260.508} C_VEL
LIN {X 0,Y 533.642,Z 721.051,A -85,B 0,C 180,E1 23260.007,E2 23260.007} C_VEL
LIN {X 0,Y 521.927,Z 796.054,A -85,B 0,C 180,E1 23258.09,E2 23258.09} C_VEL
LIN {X 0,Y 512.951,Z 867.575,A -85,B 0,C 180,E1 23256.304,E2 23256.304} C_VEL
LIN {X 0,Y 505.082,Z 949.029,A -85,B 0,C 180,E1 23254.328,E2 23254.328} C_VEL
LIN {X 0,Y 502.709,Z 972.185,A -85,B 0,C 180,E1 23253.55,E2 23253.55} C_VEL
LIN {X 0,Y 500.094,Z 994.228,A -85,B 0,C 180,E1 23252.607,E2 23252.607} C_VEL
LIN {X 0,Y 497.065,Z 1016.812,A -85,B 0,C 180,E1 23251.402,E2 23251.402} C_VEL
LIN {X 0,Y 494.017,Z 1037.376,A -85,B 0,C 180,E1 23250.064,E2 23250.064} C_VEL
LIN {X 0,Y 490.996,Z 1056.366,A -85,B 0,C 180,E1 23248.594,E2 23248.594} C_VEL
LIN {X 0,Y 487.85,Z 1075.203,A -85,B 0,C 180,E1 23246.87,E2 23246.87} C_VEL
LIN {X 0,Y 484.96,Z 1091.917,A -85,B 0,C 180,E1 23245.071,E2 23245.071} C_VEL
LIN {X 0,Y 482.198,Z 1107.663,A -85,B 0,C 180,E1 23243.076,E2 23243.076} C_VEL
LIN {X 0,Y 479.624,Z 1122.205,A -85,B 0,C 180,E1 23240.887,E2 23240.887} C_VEL
LIN {X 0,Y 477.518,Z 1134.542,A -85,B 0,C 180,E1 23238.688,E2 23238.688} C_VEL
LIN {X 0,Y 475.765,Z 1145.547,A -85,B 0,C 180,E1 23236.359,E2 23236.359} C_VEL
LIN {X 0,Y 474.387,Z 1155.128,A -85,B 0,C 180,E1 23233.906,E2 23233.906} C_VEL
LIN {X 0,Y 473.392,Z 1162.748,A -85,B 0,C 180,E1 23231.454,E2 23231.454} C_VEL
LIN {X 0,Y 472.735,Z 1168.982,A -85,B 0,C 180,E1 23228.885,E2 23228.885} C_VEL
LIN {X 0,Y 472.376,Z 1173.348,A -85,B 0,C 180,E1 23226.444,E2 23226.444} C_VEL
LIN {X 0,Y 472.176,Z 1176.178,A -85,B 0,C 180,E1 23223.888,E2 23223.888} C_VEL
LIN {X 0,Y 472.102,Z 1177.452,A -85,B 0,C 180,E1 23221.216,E2 23221.216} C_VEL
LIN {X 0,Y 472.077,Z 1177.076,A -85,B 0,C 180,E1 23218.689,E2 23218.689} C_VEL
LIN {X 0,Y 472.1,Z 1175.093,A -85,B 0,C 180,E1 23216.238,E2 23216.238} C_VEL
LIN {X 0,Y 472.208,Z 1171.444,A -85,B 0,C 180,E1 23213.681,E2 23213.681} C_VEL
LIN {X 0,Y 472.471,Z 1166.424,A -85,B 0,C 180,E1 23211.235,E2 23211.235} C_VEL
LIN {X 0,Y 472.93,Z 1159.635,A -85,B 0,C 180,E1 23208.787,E2 23208.787} C_VEL
LIN {X 0,Y 473.692,Z 1151.09,A -85,B 0,C 180,E1 23206.328,E2 23206.328} C_VEL
LIN {X 0,Y 474.759,Z 1141.194,A -85,B 0,C 180,E1 23203.987,E2 23203.987} C_VEL
LIN {X 0,Y 476.118,Z 1129.883,A -85,B 0,C 180,E1 23201.768,E2 23201.768} C_VEL
LIN {X 0,Y 477.858,Z 1116.512,A -85,B 0,C 180,E1 23199.55,E2 23199.55} C_VEL
LIN {X 0,Y 479.959,Z 1101.195,A -85,B 0,C 180,E1 23197.399,E2 23197.399} C_VEL
LIN {X 0,Y 482.173,Z 1085.349,A -85,B 0,C 180,E1 23195.5,E2 23195.5} C_VEL
LIN {X 0,Y 484.554,Z 1067.923,A -85,B 0,C 180,E1 23193.732,E2 23193.732} C_VEL
LIN {X 0,Y 486.953,Z 1049.639,A -85,B 0,C 180,E1 23192.155,E2 23192.155} C_VEL
LIN {X 0,Y 489.504,Z 1028.896,A -85,B 0,C 180,E1 23190.647,E2 23190.647} C_VEL
LIN {X 0,Y 491.745,Z 1009.147,A -85,B 0,C 180,E1 23189.451,E2 23189.451} C_VEL
LIN {X 0,Y 493.902,Z 987.457,A -85,B 0,C 180,E1 23188.38,E2 23188.38} C_VEL
LIN {X 0,Y 495.711,Z 965.46,A -85,B 0,C 180,E1 23187.522,E2 23187.522} C_VEL
LIN {X 0,Y 497.246,Z 942.245,A -85,B 0,C 180,E1 23186.837,E2 23186.837} C_VEL
LIN {X 0,Y 498.511,Z 915.865,A -85,B 0,C 180,E1 23186.3,E2 23186.3} C_VEL
LIN {X 0,Y 507.676,Z 701.576,A -85,B 0,C 180,E1 23182.509,E2 23182.509} C_VEL
LIN {X 0,Y 488.008,Z 666.387,A -85,B 0,C 180,E1 23180.23,E2 23180.23} C_VEL
LIN {X 0,Y 475.584,Z 645.326,A -85,B 0,C 180,E1 23178.71,E2 23178.71} C_VEL
LIN {X 0,Y 474.164,Z 641.935,A -85,B 0,C 180,E1 23178.505,E2 23178.505} C_VEL
LIN {X 0,Y 474.117,Z 641.605,A -85,B 0,C 180,E1 23178.477,E2 23178.477} C_VEL
LIN {X 0,Y 474.084,Z 641.612,A -85,B 0,C 180,E1 23174.879,E2 23174.879} C_VEL
LIN {X 0,Y 474.053,Z 641.62,A -85,B 0,C 180,E1 23171.316,E2 23171.316} C_VEL
LIN {X 0,Y 474.082,Z 641.611,A -85,B 0,C 180,E1 23167.862,E2 23167.862} C_VEL
LIN {X 0,Y 474.115,Z 641.612,A -85,B 0,C 180,E1 23164.244,E2 23164.244} C_VEL
LIN {X 0,Y 474.11,Z 641.611,A -85,B 0,C 180,E1 23160.55,E2 23160.55} C_VEL
LIN {X 0,Y 474.1,Z 641.612,A -85,B 0,C 180,E1 23156.966,E2 23156.966} C_VEL
LIN {X 0,Y 474.091,Z 641.614,A -85,B 0,C 180,E1 23153.361,E2 23153.361} C_VEL
LIN {X 0,Y 474.093,Z 641.615,A -85,B 0,C 180,E1 23149.723,E2 23149.723} C_VEL
LIN {X 0,Y 474.098,Z 641.613,A -85,B 0,C 180,E1 23146.166,E2 23146.166} C_VEL
LIN {X 0,Y 474.106,Z 641.604,A -85,B 0,C 180,E1 23142.548,E2 23142.548} C_VEL
LIN {X 0,Y 474.116,Z 641.601,A -85,B 0,C 180,E1 23138.858,E2 23138.858} C_VEL
LIN {X 0,Y 474.084,Z 641.615,A -85,B 0,C 180,E1 23135.326,E2 23135.326} C_VEL
LIN {X 0,Y 474.053,Z 641.605,A -85,B 0,C 180,E1 23131.694,E2 23131.694} C_VEL
LIN {X 0,Y 474.104,Z 641.607,A -85,B 0,C 180,E1 23131.09,E2 23131.09} C_VEL
LIN {X 0,Y 473.152,Z 641.737,A -85,B 0,C 180,E1 23130.159,E2 23130.159} C_VEL
LIN {X 0,Y 466.622,Z 642.536,A -85,B 0,C 180,E1 23127.474,E2 23127.474} C_VEL
LIN {X 0,Y 466.167,Z 642.585,A -85,B 0,C 180,E1 23126.858,E2 23126.858} C_VEL
LIN {X 0,Y 466.163,Z 642.598,A -85,B 0,C 180,E1 23123.227,E2 23123.227} C_VEL
LIN {X 0,Y 466.131,Z 642.587,A -85,B 0,C 180,E1 23119.621,E2 23119.621} C_VEL
LIN {X 0,Y 466.108,Z 642.605,A -85,B 0,C 180,E1 23115.973,E2 23115.973} C_VEL
LIN {X 0,Y 466.156,Z 642.6,A -85,B 0,C 180,E1 23112.398,E2 23112.398} C_VEL
LIN {X 0,Y 466.18,Z 642.599,A -85,B 0,C 180,E1 23108.75,E2 23108.75} C_VEL
LIN {X 0,Y 466.164,Z 642.6,A -85,B 0,C 180,E1 23105.126,E2 23105.126} C_VEL
LIN {X 0,Y 466.153,Z 642.603,A -85,B 0,C 180,E1 23101.566,E2 23101.566} C_VEL
LIN {X 0,Y 466.15,Z 642.604,A -85,B 0,C 180,E1 23098.01,E2 23098.01} C_VEL
LIN {X 0,Y 466.161,Z 642.603,A -85,B 0,C 180,E1 23094.311,E2 23094.311} C_VEL
LIN {X 0,Y 466.169,Z 642.601,A -85,B 0,C 180,E1 23090.737,E2 23090.737} C_VEL
LIN {X 0,Y 466.172,Z 642.595,A -85,B 0,C 180,E1 23087.165,E2 23087.165} C_VEL
LIN {X 0,Y 466.185,Z 642.754,A -85,B 0,C 180,E1 23086.792,E2 23086.792} C_VEL
LIN {X 0,Y 474.387,Z 670.11,A -85,B 0,C 180,E1 23083.879,E2 23083.879} C_VEL
LIN {X 0,Y 478.757,Z 687.054,A -85,B 0,C 180,E1 23082.151,E2 23082.151} C_VEL
LIN {X 0,Y 476.977,Z 730.678,A -85,B 0,C 180,E1 23078.435,E2 23078.435} C_VEL
LIN {X 0,Y 475.28,Z 771.673,A -85,B 0,C 180,E1 23074.961,E2 23074.961} C_VEL
LIN {X 0,Y 473.647,Z 814.343,A -85,B 0,C 180,E1 23071.36,E2 23071.36} C_VEL
LIN {X 0,Y 472.778,Z 839.653,A -85,B 0,C 180,E1 23069.266,E2 23069.266} C_VEL
LIN {X 0,Y 470.192,Z 982.916,A -85,B 0,C 180,E1 23066.589,E2 23066.589} C_VEL
LIN {X 0,Y 469.961,Z 999.291,A -85,B 0,C 180,E1 23066.077,E2 23066.077} C_VEL
LIN {X 0,Y 469.517,Z 1015.604,A -85,B 0,C 180,E1 23065.34,E2 23065.34} C_VEL
LIN {X 0,Y 468.984,Z 1030.571,A -85,B 0,C 180,E1 23064.429,E2 23064.429} C_VEL
LIN {X 0,Y 468.36,Z 1044.792,A -85,B 0,C 180,E1 23063.328,E2 23063.328} C_VEL
LIN {X 0,Y 467.681,Z 1058.005,A -85,B 0,C 180,E1 23062.034,E2 23062.034} C_VEL
LIN {X 0,Y 467.077,Z 1069.257,A -85,B 0,C 180,E1 23060.681,E2 23060.681} C_VEL
LIN {X 0,Y 466.5,Z 1079.562,A -85,B 0,C 180,E1 23059.14,E2 23059.14} C_VEL
LIN {X 0,Y 466.043,Z 1088.495,A -85,B 0,C 180,E1 23057.477,E2 23057.477} C_VEL
LIN {X 0,Y 465.712,Z 1095.885,A -85,B 0,C 180,E1 23055.692,E2 23055.692} C_VEL
LIN {X 0,Y 465.516,Z 1101.746,A -85,B 0,C 180,E1 23053.79,E2 23053.79} C_VEL
LIN {X 0,Y 465.46,Z 1106.001,A -85,B 0,C 180,E1 23051.647,E2 23051.647} C_VEL
LIN {X 0,Y 465.555,Z 1107.897,A -85,B 0,C 180,E1 23049.766,E2 23049.766} C_VEL
LIN {X 0,Y 465.794,Z 1108.026,A -85,B 0,C 180,E1 23047.77,E2 23047.77} C_VEL
LIN {X 0,Y 466.182,Z 1106.433,A -85,B 0,C 180,E1 23045.906,E2 23045.906} C_VEL
LIN {X 0,Y 466.764,Z 1102.797,A -85,B 0,C 180,E1 23043.928,E2 23043.928} C_VEL
LIN {X 0,Y 467.51,Z 1097.517,A -85,B 0,C 180,E1 23042.081,E2 23042.081} C_VEL
LIN {X 0,Y 468.466,Z 1090.163,A -85,B 0,C 180,E1 23040.242,E2 23040.242} C_VEL
LIN {X 0,Y 469.483,Z 1081.874,A -85,B 0,C 180,E1 23038.655,E2 23038.655} C_VEL
LIN {X 0,Y 470.663,Z 1071.414,A -85,B 0,C 180,E1 23037.075,E2 23037.075} C_VEL
LIN {X 0,Y 471.822,Z 1059.793,A -85,B 0,C 180,E1 23035.683,E2 23035.683} C_VEL
LIN {X 0,Y 472.943,Z 1046.525,A -85,B 0,C 180,E1 23034.417,E2 23034.417} C_VEL
LIN {X 0,Y 473.847,Z 1032.908,A -85,B 0,C 180,E1 23033.394,E2 23033.394} C_VEL
LIN {X 0,Y 474.537,Z 1019.526,A -85,B 0,C 180,E1 23032.613,E2 23032.613} C_VEL
LIN {X 0,Y 475.055,Z 1006.653,A -85,B 0,C 180,E1 23032.02,E2 23032.02} C_VEL
LIN {X 0,Y 475.425,Z 991.878,A -85,B 0,C 180,E1 23031.509,E2 23031.509} C_VEL
LIN {X 0,Y 476.138,Z 953.559,A -85,B 0,C 180,E1 23030.692,E2 23030.692} C_VEL
LIN {X 0,Y 480.232,Z 850.632,A -85,B 0,C 180,E1 23028.559,E2 23028.559} C_VEL
LIN {X 0,Y 480.749,Z 847.244,A -85,B 0,C 180,E1 23028.298,E2 23028.298} C_VEL
LIN {X 0,Y 483.282,Z 801.014,A -85,B 0,C 180,E1 23024.395,E2 23024.395} C_VEL
LIN {X 0,Y 485.64,Z 758.484,A -85,B 0,C 180,E1 23020.826,E2 23020.826} C_VEL
LIN {X 0,Y 488.117,Z 716.796,A -85,B 0,C 180,E1 23017.347,E2 23017.347} C_VEL
LIN {X 0,Y 489.327,Z 696.184,A -85,B 0,C 180,E1 23015.619,E2 23015.619} C_VEL
LIN {X 0,Y 485.846,Z 684.137,A -85,B 0,C 180,E1 23014.069,E2 23014.069} C_VEL
LIN {X 0,Y 481.2,Z 671.86,A -85,B 0,C 180,E1 23012.258,E2 23012.258} C_VEL
LIN {X 0,Y 476.385,Z 661.441,A -85,B 0,C 180,E1 23010.444,E2 23010.444} C_VEL
LIN {X 0,Y 473.717,Z 656.447,A -85,B 0,C 180,E1 23009.444,E2 23009.444} C_VEL
LIN {X 0,Y 471.751,Z 652.655,A -85,B 0,C 180,E1 23008.663,E2 23008.663} C_VEL
LIN {X 0,Y 469.722,Z 649.232,A -85,B 0,C 180,E1 23007.845,E2 23007.845} C_VEL
LIN {X 0,Y 469.121,Z 647.865,A -85,B 0,C 180,E1 23007.565,E2 23007.565} C_VEL
LIN {X 0,Y 466.766,Z 644.855,A -85,B 0,C 180,E1 23006.658,E2 23006.658} C_VEL
LIN {X 0,Y 466.161,Z 642.601,A -85,B 0,C 180,E1 23006.186,E2 23006.186} C_VEL
LIN {X 0,Y 466.141,Z 642.605,A -85,B 0,C 180,E1 23002.525,E2 23002.525} C_VEL
LIN {X 0,Y 466.163,Z 642.6,A -85,B 0,C 180,E1 22999.023,E2 22999.023} C_VEL
LIN {X 0,Y 466.178,Z 642.663,A -85,B 0,C 180,E1 22996.541,E2 22996.541} C_VEL
LIN {X 0,Y 473.813,Z 665.298,A -85,B 0,C 180,E1 22992.92,E2 22992.92} C_VEL
LIN {X 0,Y 477.155,Z 675.381,A -85,B 0,C 180,E1 22991.427,E2 22991.427} C_VEL
LIN {X 0,Y 494.551,Z 709.83,A -85,B 0,C 180,E1 22989.228,E2 22989.228} C_VEL
LIN {X 0,Y 497.709,Z 716.98,A -85,B 0,C 180,E1 22988.83,E2 22988.83} C_VEL
LIN {X 0,Y 500.884,Z 736.059,A -85,B 0,C 180,E1 22988.175,E2 22988.175} C_VEL
LIN {X 0,Y 489.837,Z 981.437,A -85,B 0,C 180,E1 22983.697,E2 22983.697} C_VEL
LIN {X 0,Y 488.076,Z 1005.008,A -85,B 0,C 180,E1 22983.056,E2 22983.056} C_VEL
LIN {X 0,Y 486.126,Z 1026.44,A -85,B 0,C 180,E1 22982.264,E2 22982.264} C_VEL
LIN {X 0,Y 483.812,Z 1048.241,A -85,B 0,C 180,E1 22981.245,E2 22981.245} C_VEL
LIN {X 0,Y 481.344,Z 1069.167,A -85,B 0,C 180,E1 22980.039,E2 22980.039} C_VEL
LIN {X 0,Y 478.724,Z 1089.669,A -85,B 0,C 180,E1 22978.608,E2 22978.608} C_VEL
LIN {X 0,Y 476.156,Z 1108.413,A -85,B 0,C 180,E1 22977.039,E2 22977.039} C_VEL
LIN {X 0,Y 473.713,Z 1126.034,A -85,B 0,C 180,E1 22975.307,E2 22975.307} C_VEL
LIN {X 0,Y 471.439,Z 1142.382,A -85,B 0,C 180,E1 22973.431,E2 22973.431} C_VEL
LIN {X 0,Y 469.373,Z 1157.76,A -85,B 0,C 180,E1 22971.361,E2 22971.361} C_VEL
LIN {X 0,Y 467.663,Z 1171.211,A -85,B 0,C 180,E1 22969.222,E2 22969.222} C_VEL
LIN {X 0,Y 466.222,Z 1183.969,A -85,B 0,C 180,E1 22966.828,E2 22966.828} C_VEL
LIN {X 0,Y 465.206,Z 1194.642,A -85,B 0,C 180,E1 22964.436,E2 22964.436} C_VEL
LIN {X 0,Y 464.558,Z 1203.364,A -85,B 0,C 180,E1 22962.049,E2 22962.049} C_VEL
LIN {X 0,Y 464.191,Z 1210.669,A -85,B 0,C 180,E1 22959.545,E2 22959.545} C_VEL
LIN {X 0,Y 464.057,Z 1216.271,A -85,B 0,C 180,E1 22957.053,E2 22957.053} C_VEL
LIN {X 0,Y 464.044,Z 1219.957,A -85,B 0,C 180,E1 22954.695,E2 22954.695} C_VEL
LIN {X 0,Y 464.085,Z 1222.373,A -85,B 0,C 180,E1 22952.097,E2 22952.097} C_VEL
LIN {X 0,Y 464.086,Z 1223.075,A -85,B 0,C 180,E1 22949.751,E2 22949.751} C_VEL
LIN {X 0,Y 464.058,Z 1222.208,A -85,B 0,C 180,E1 22947.281,E2 22947.281} C_VEL
LIN {X 0,Y 464.018,Z 1219.854,A -85,B 0,C 180,E1 22944.806,E2 22944.806} C_VEL
LIN {X 0,Y 464.053,Z 1215.787,A -85,B 0,C 180,E1 22942.321,E2 22942.321} C_VEL
LIN {X 0,Y 464.265,Z 1209.8,A -85,B 0,C 180,E1 22939.701,E2 22939.701} C_VEL
LIN {X 0,Y 464.746,Z 1202.363,A -85,B 0,C 180,E1 22937.195,E2 22937.195} C_VEL
LIN {X 0,Y 465.539,Z 1193.448,A -85,B 0,C 180,E1 22934.808,E2 22934.808} C_VEL
LIN {X 0,Y 466.827,Z 1182.142,A -85,B 0,C 180,E1 22932.292,E2 22932.292} C_VEL
LIN {X 0,Y 468.443,Z 1170.079,A -85,B 0,C 180,E1 22930.029,E2 22930.029} C_VEL
LIN {X 0,Y 470.535,Z 1155.785,A -85,B 0,C 180,E1 22927.773,E2 22927.773} C_VEL
LIN {X 0,Y 473.012,Z 1140.045,A -85,B 0,C 180,E1 22925.655,E2 22925.655} C_VEL
LIN {X 0,Y 475.903,Z 1122.317,A -85,B 0,C 180,E1 22923.616,E2 22923.616} C_VEL
LIN {X 0,Y 479.037,Z 1103.598,A -85,B 0,C 180,E1 22921.784,E2 22921.784} C_VEL
LIN {X 0,Y 482.388,Z 1083.26,A -85,B 0,C 180,E1 22920.097,E2 22920.097} C_VEL
LIN {X 0,Y 485.802,Z 1061.978,A -85,B 0,C 180,E1 22918.617,E2 22918.617} C_VEL
LIN {X 0,Y 489.202,Z 1039.987,A -85,B 0,C 180,E1 22917.343,E2 22917.343} C_VEL
LIN {X 0,Y 492.568,Z 1017.048,A -85,B 0,C 180,E1 22916.253,E2 22916.253} C_VEL
LIN {X 0,Y 495.854,Z 992.946,A -85,B 0,C 180,E1 22915.342,E2 22915.342} C_VEL
LIN {X 0,Y 498.871,Z 967.405,A -85,B 0,C 180,E1 22914.601,E2 22914.601} C_VEL
LIN {X 0,Y 507.071,Z 886.457,A -85,B 0,C 180,E1 22912.633,E2 22912.633} C_VEL
LIN {X 0,Y 516.463,Z 814.164,A -85,B 0,C 180,E1 22910.788,E2 22910.788} C_VEL
LIN {X 0,Y 528.228,Z 740.621,A -85,B 0,C 180,E1 22908.875,E2 22908.875} C_VEL
LIN {X 0,Y 528.663,Z 734.478,A -85,B 0,C 180,E1 22908.504,E2 22908.504} C_VEL
LIN {X 0,Y 527.521,Z 729.171,A -85,B 0,C 180,E1 22907.543,E2 22907.543} C_VEL
LIN {X 0,Y 526.668,Z 724.865,A -85,B 0,C 180,E1 22906.49,E2 22906.49} C_VEL
LIN {X 0,Y 526.149,Z 722.085,A -85,B 0,C 180,E1 22905.298,E2 22905.298} C_VEL
LIN {X 0,Y 526.341,Z 720.575,A -85,B 0,C 180,E1 22904.102,E2 22904.102} C_VEL
LIN {X 0,Y 527.478,Z 721.059,A -85,B 0,C 180,E1 22902.591,E2 22902.591} C_VEL
LIN {X 0,Y 528.998,Z 723.875,A -85,B 0,C 180,E1 22901.374,E2 22901.374} C_VEL
LIN {X 0,Y 530.124,Z 726.295,A -85,B 0,C 180,E1 22900.7,E2 22900.7} C_VEL
LIN {X 0,Y 517.675,Z 799.906,A -85,B 0,C 180,E1 22898.783,E2 22898.783} C_VEL
LIN {X 0,Y 508.181,Z 869.083,A -85,B 0,C 180,E1 22897.008,E2 22897.008} C_VEL
LIN {X 0,Y 499.522,Z 950.022,A -85,B 0,C 180,E1 22894.974,E2 22894.974} C_VEL
LIN {X 0,Y 496.874,Z 973.534,A -85,B 0,C 180,E1 22894.158,E2 22894.158} C_VEL
LIN {X 0,Y 494.047,Z 995.412,A -85,B 0,C 180,E1 22893.195,E2 22893.195} C_VEL
LIN {X 0,Y 490.692,Z 1018.563,A -85,B 0,C 180,E1 22891.926,E2 22891.926} C_VEL
LIN {X 0,Y 487.341,Z 1039.623,A -85,B 0,C 180,E1 22890.516,E2 22890.516} C_VEL
LIN {X 0,Y 484.044,Z 1058.859,A -85,B 0,C 180,E1 22888.976,E2 22888.976} C_VEL
LIN {X 0,Y 480.847,Z 1076.685,A -85,B 0,C 180,E1 22887.294,E2 22887.294} C_VEL
LIN {X 0,Y 477.799,Z 1093.178,A -85,B 0,C 180,E1 22885.473,E2 22885.473} C_VEL
LIN {X 0,Y 474.887,Z 1108.788,A -85,B 0,C 180,E1 22883.452,E2 22883.452} C_VEL
LIN {X 0,Y 472.164,Z 1123.205,A -85,B 0,C 180,E1 22881.233,E2 22881.233} C_VEL
LIN {X 0,Y 469.927,Z 1135.43,A -85,B 0,C 180,E1 22879.001,E2 22879.001} C_VEL
LIN {X 0,Y 467.972,Z 1146.852,A -85,B 0,C 180,E1 22876.512,E2 22876.512} C_VEL
LIN {X 0,Y 466.522,Z 1156.269,A -85,B 0,C 180,E1 22874.018,E2 22874.018} C_VEL
LIN {X 0,Y 465.48,Z 1163.774,A -85,B 0,C 180,E1 22871.526,E2 22871.526} C_VEL
LIN {X 0,Y 464.807,Z 1169.588,A -85,B 0,C 180,E1 22869.037,E2 22869.037} C_VEL
LIN {X 0,Y 464.417,Z 1173.9,A -85,B 0,C 180,E1 22866.555,E2 22866.555} C_VEL
LIN {X 0,Y 464.203,Z 1176.575,A -85,B 0,C 180,E1 22864.079,E2 22864.079} C_VEL
LIN {X 0,Y 464.117,Z 1177.876,A -85,B 0,C 180,E1 22861.361,E2 22861.361} C_VEL
LIN {X 0,Y 464.09,Z 1177.569,A -85,B 0,C 180,E1 22858.892,E2 22858.892} C_VEL
LIN {X 0,Y 464.106,Z 1175.657,A -85,B 0,C 180,E1 22856.421,E2 22856.421} C_VEL
LIN {X 0,Y 464.209,Z 1172.112,A -85,B 0,C 180,E1 22853.82,E2 22853.82} C_VEL
LIN {X 0,Y 464.466,Z 1167.144,A -85,B 0,C 180,E1 22851.336,E2 22851.336} C_VEL
LIN {X 0,Y 464.93,Z 1160.435,A -85,B 0,C 180,E1 22848.843,E2 22848.843} C_VEL
LIN {X 0,Y 465.749,Z 1151.504,A -85,B 0,C 180,E1 22846.217,E2 22846.217} C_VEL
LIN {X 0,Y 466.854,Z 1141.589,A -85,B 0,C 180,E1 22843.837,E2 22843.837} C_VEL
LIN {X 0,Y 468.26,Z 1130.247,A -85,B 0,C 180,E1 22841.58,E2 22841.58} C_VEL
LIN {X 0,Y 470.06,Z 1116.842,A -85,B 0,C 180,E1 22839.326,E2 22839.326} C_VEL
LIN {X 0,Y 472.165,Z 1101.964,A -85,B 0,C 180,E1 22837.202,E2 22837.202} C_VEL
LIN {X 0,Y 474.432,Z 1086.219,A -85,B 0,C 180,E1 22835.281,E2 22835.281} C_VEL
LIN {X 0,Y 476.886,Z 1068.743,A -85,B 0,C 180,E1 22833.478,E2 22833.478} C_VEL
LIN {X 0,Y 479.35,Z 1050.521,A -85,B 0,C 180,E1 22831.877,E2 22831.877} C_VEL
LIN {X 0,Y 481.903,Z 1030.459,A -85,B 0,C 180,E1 22830.387,E2 22830.387} C_VEL
LIN {X 0,Y 484.273,Z 1010.267,A -85,B 0,C 180,E1 22829.134,E2 22829.134} C_VEL
LIN {X 0,Y 486.48,Z 988.7,A -85,B 0,C 180,E1 22828.049,E2 22828.049} C_VEL
LIN {X 0,Y 488.366,Z 966.769,A -85,B 0,C 180,E1 22827.17,E2 22827.17} C_VEL
LIN {X 0,Y 489.992,Z 943.094,A -85,B 0,C 180,E1 22826.452,E2 22826.452} C_VEL
LIN {X 0,Y 491.242,Z 918.549,A -85,B 0,C 180,E1 22825.934,E2 22825.934} C_VEL
LIN {X 0,Y 500.837,Z 704.44,A -85,B 0,C 180,E1 22822.074,E2 22822.074} C_VEL
LIN {X 0,Y 482.128,Z 670.923,A -85,B 0,C 180,E1 22819.863,E2 22819.863} C_VEL
LIN {X 0,Y 467.775,Z 646.491,A -85,B 0,C 180,E1 22818.063,E2 22818.063} C_VEL
LIN {X 0,Y 466.25,Z 643.102,A -85,B 0,C 180,E1 22817.842,E2 22817.842} C_VEL
LIN {X 0,Y 466.171,Z 642.597,A -85,B 0,C 180,E1 22817.792,E2 22817.792} C_VEL
LIN {X 0,Y 466.172,Z 642.597,A -85,B 0,C 180,E1 22814.195,E2 22814.195} C_VEL
LIN {X 0,Y 466.116,Z 642.607,A -85,B 0,C 180,E1 22810.704,E2 22810.704} C_VEL
LIN {X 0,Y 466.113,Z 642.605,A -85,B 0,C 180,E1 22807.066,E2 22807.066} C_VEL
LIN {X 0,Y 466.15,Z 642.601,A -85,B 0,C 180,E1 22803.453,E2 22803.453} C_VEL
LIN {X 0,Y 466.182,Z 642.595,A -85,B 0,C 180,E1 22799.843,E2 22799.843} C_VEL
LIN {X 0,Y 466.145,Z 642.598,A -85,B 0,C 180,E1 22796.225,E2 22796.225} C_VEL
LIN {X 0,Y 466.1,Z 642.602,A -85,B 0,C 180,E1 22792.583,E2 22792.583} C_VEL
LIN {X 0,Y 466.119,Z 642.601,A -85,B 0,C 180,E1 22788.901,E2 22788.901} C_VEL
LIN {X 0,Y 466.167,Z 642.597,A -85,B 0,C 180,E1 22785.299,E2 22785.299} C_VEL
LIN {X 0,Y 466.166,Z 642.599,A -85,B 0,C 180,E1 22781.633,E2 22781.633} C_VEL
LIN {X 0,Y 466.136,Z 642.595,A -85,B 0,C 180,E1 22778.016,E2 22778.016} C_VEL
LIN {X 0,Y 466.108,Z 642.603,A -85,B 0,C 180,E1 22774.431,E2 22774.431} C_VEL
LIN {X 0,Y 466.14,Z 642.602,A -85,B 0,C 180,E1 22770.739,E2 22770.739} C_VEL
LIN {X 0,Y 466.175,Z 642.586,A -85,B 0,C 180,E1 22767.174,E2 22767.174} C_VEL
LIN {X 0,Y 466.167,Z 642.585,A -85,B 0,C 180,E1 22766.858,E2 22766.858} C_VEL
LIN {X 0,Y 465.163,Z 642.71,A -85,B 0,C 180,E1 22765.912,E2 22765.912} C_VEL
LIN {X 0,Y 458.679,Z 643.532,A -85,B 0,C 180,E1 22763.178,E2 22763.178} C_VEL
LIN {X 0,Y 458.241,Z 643.586,A -85,B 0,C 180,E1 22762.552,E2 22762.552} C_VEL
LIN {X 0,Y 458.208,Z 643.571,A -85,B 0,C 180,E1 22758.931,E2 22758.931} C_VEL
LIN {X 0,Y 458.16,Z 643.594,A -85,B 0,C 180,E1 22755.338,E2 22755.338} C_VEL
LIN {X 0,Y 458.19,Z 643.591,A -85,B 0,C 180,E1 22751.662,E2 22751.662} C_VEL
LIN {X 0,Y 458.219,Z 643.589,A -85,B 0,C 180,E1 22747.958,E2 22747.958} C_VEL
LIN {X 0,Y 458.237,Z 643.585,A -85,B 0,C 180,E1 22744.266,E2 22744.266} C_VEL
LIN {X 0,Y 458.19,Z 643.593,A -85,B 0,C 180,E1 22740.739,E2 22740.739} C_VEL
LIN {X 0,Y 458.161,Z 643.597,A -85,B 0,C 180,E1 22737.086,E2 22737.086} C_VEL
LIN {X 0,Y 458.196,Z 643.592,A -85,B 0,C 180,E1 22733.417,E2 22733.417} C_VEL
LIN {X 0,Y 458.236,Z 643.587,A -85,B 0,C 180,E1 22729.771,E2 22729.771} C_VEL
LIN {X 0,Y 458.268,Z 643.83,A -85,B 0,C 180,E1 22727.194,E2 22727.194} C_VEL
LIN {X 0,Y 466.408,Z 670.755,A -85,B 0,C 180,E1 22724.276,E2 22724.276} C_VEL
LIN {X 0,Y 471.243,Z 688.838,A -85,B 0,C 180,E1 22722.409,E2 22722.409} C_VEL
LIN {X 0,Y 469.405,Z 732.171,A -85,B 0,C 180,E1 22718.692,E2 22718.692} C_VEL
LIN {X 0,Y 467.626,Z 773.071,A -85,B 0,C 180,E1 22715.191,E2 22715.191} C_VEL
LIN {X 0,Y 465.934,Z 815.606,A -85,B 0,C 180,E1 22711.572,E2 22711.572} C_VEL
LIN {X 0,Y 465.05,Z 840.421,A -85,B 0,C 180,E1 22709.503,E2 22709.503} C_VEL
LIN {X 0,Y 462.337,Z 983.861,A -85,B 0,C 180,E1 22706.76,E2 22706.76} C_VEL
LIN {X 0,Y 462.091,Z 1000.546,A -85,B 0,C 180,E1 22706.226,E2 22706.226} C_VEL
LIN {X 0,Y 461.62,Z 1017.178,A -85,B 0,C 180,E1 22705.455,E2 22705.455} C_VEL
LIN {X 0,Y 461.04,Z 1032.828,A -85,B 0,C 180,E1 22704.468,E2 22704.468} C_VEL
LIN {X 0,Y 460.397,Z 1046.771,A -85,B 0,C 180,E1 22703.347,E2 22703.347} C_VEL
LIN {X 0,Y 459.682,Z 1060.405,A -85,B 0,C 180,E1 22701.967,E2 22701.967} C_VEL
LIN {X 0,Y 459.035,Z 1071.918,A -85,B 0,C 180,E1 22700.512,E2 22700.512} C_VEL
LIN {X 0,Y 458.434,Z 1082.693,A -85,B 0,C 180,E1 22698.817,E2 22698.817} C_VEL
LIN {X 0,Y 457.98,Z 1091.644,A -85,B 0,C 180,E1 22697.008,E2 22697.008} C_VEL
LIN {X 0,Y 457.691,Z 1098.562,A -85,B 0,C 180,E1 22695.195,E2 22695.195} C_VEL
LIN {X 0,Y 457.524,Z 1103.517,A -85,B 0,C 180,E1 22693.392,E2 22693.392} C_VEL
LIN {X 0,Y 457.515,Z 1107.151,A -85,B 0,C 180,E1 22691.468,E2 22691.468} C_VEL
LIN {X 0,Y 457.628,Z 1108.945,A -85,B 0,C 180,E1 22689.556,E2 22689.556} C_VEL
LIN {X 0,Y 457.91,Z 1109.014,A -85,B 0,C 180,E1 22687.525,E2 22687.525} C_VEL
